LIN {X 0,Y 375.979,Z 740.463,A -85,B 0,C 180,E1 -12485.717,E2 -12485.717} C_VEL
LIN {X 0,Y 376.052,Z 740.601,A -85,B 0,C 180,E1 -12488.619,E2 -12488.619} C_VEL
LIN {X 0,Y 376.894,Z 745.86,A -85,B 0,C 180,E1 -12490.388,E2 -12490.388} C_VEL
LIN {X 0,Y 376.824,Z 753.026,A -85,B 0,C 180,E1 -12492.638,E2 -12492.638} C_VEL
LIN {X 0,Y 376.652,Z 755.465,A -85,B 0,C 180,E1 -12493.328,E2 -12493.328} C_VEL
LIN {X 0,Y 377.194,Z 758.566,A -85,B 0,C 180,E1 -12493.474,E2 -12493.474} C_VEL
LIN {X 0,Y 380.294,Z 775.584,A -85,B 0,C 180,E1 -12493.943,E2 -12493.943} C_VEL
LIN {X 0,Y 379.732,Z 831.118,A -85,B 0,C 180,E1 -12495.017,E2 -12495.017} C_VEL
LIN {X 0,Y 379.481,Z 840.948,A -85,B 0,C 180,E1 -12495.35,E2 -12495.35} C_VEL
LIN {X 0,Y 378.941,Z 852.061,A -85,B 0,C 180,E1 -12495.911,E2 -12495.911} C_VEL
LIN {X 0,Y 378.37,Z 862.886,A -85,B 0,C 180,E1 -12496.711,E2 -12496.711} C_VEL
LIN {X 0,Y 377.773,Z 871.277,A -85,B 0,C 180,E1 -12497.51,E2 -12497.51} C_VEL
LIN {X 0,Y 377.216,Z 879.195,A -85,B 0,C 180,E1 -12498.446,E2 -12498.446} C_VEL
LIN {X 0,Y 376.73,Z 884.882,A -85,B 0,C 180,E1 -12499.248,E2 -12499.248} C_VEL
LIN {X 0,Y 376.171,Z 891.229,A -85,B 0,C 180,E1 -12500.32,E2 -12500.32} C_VEL
LIN {X 0,Y 375.646,Z 897.671,A -85,B 0,C 180,E1 -12501.663,E2 -12501.663} C_VEL
LIN {X 0,Y 375.314,Z 902.635,A -85,B 0,C 180,E1 -12502.96,E2 -12502.96} C_VEL
LIN {X 0,Y 374.956,Z 907.561,A -85,B 0,C 180,E1 -12504.622,E2 -12504.622} C_VEL
LIN {X 0,Y 374.741,Z 909.88,A -85,B 0,C 180,E1 -12505.698,E2 -12505.698} C_VEL
LIN {X 0,Y 374.627,Z 911.643,A -85,B 0,C 180,E1 -12506.774,E2 -12506.774} C_VEL
LIN {X 0,Y 374.591,Z 912.912,A -85,B 0,C 180,E1 -12507.85,E2 -12507.85} C_VEL
LIN {X 0,Y 374.546,Z 913.715,A -85,B 0,C 180,E1 -12508.925,E2 -12508.925} C_VEL
LIN {X 0,Y 374.553,Z 914.02,A -85,B 0,C 180,E1 -12510,E2 -12510} C_VEL
LIN {X 0,Y 374.545,Z 913.744,A -85,B 0,C 180,E1 -12511.075,E2 -12511.075} C_VEL
LIN {X 0,Y 374.577,Z 913,A -85,B 0,C 180,E1 -12512.151,E2 -12512.151} C_VEL
LIN {X 0,Y 374.626,Z 911.789,A -85,B 0,C 180,E1 -12513.226,E2 -12513.226} C_VEL
LIN {X 0,Y 374.83,Z 908.942,A -85,B 0,C 180,E1 -12514.84,E2 -12514.84} C_VEL
LIN {X 0,Y 375.043,Z 906.351,A -85,B 0,C 180,E1 -12515.916,E2 -12515.916} C_VEL
LIN {X 0,Y 375.383,Z 901.251,A -85,B 0,C 180,E1 -12517.531,E2 -12517.531} C_VEL
LIN {X 0,Y 375.802,Z 895.762,A -85,B 0,C 180,E1 -12518.875,E2 -12518.875} C_VEL
LIN {X 0,Y 376.443,Z 888.863,A -85,B 0,C 180,E1 -12520.216,E2 -12520.216} C_VEL
LIN {X 0,Y 377.105,Z 880.938,A -85,B 0,C 180,E1 -12521.421,E2 -12521.421} C_VEL
LIN {X 0,Y 377.657,Z 873.381,A -85,B 0,C 180,E1 -12522.357,E2 -12522.357} C_VEL
LIN {X 0,Y 378.109,Z 866.955,A -85,B 0,C 180,E1 -12523.025,E2 -12523.025} C_VEL
LIN {X 0,Y 378.592,Z 859.142,A -85,B 0,C 180,E1 -12523.691,E2 -12523.691} C_VEL
LIN {X 0,Y 379.141,Z 850.18,A -85,B 0,C 180,E1 -12524.286,E2 -12524.286} C_VEL
LIN {X 0,Y 379.49,Z 840.834,A -85,B 0,C 180,E1 -12524.753,E2 -12524.753} C_VEL
LIN {X 0,Y 379.72,Z 831.346,A -85,B 0,C 180,E1 -12525.076,E2 -12525.076} C_VEL
LIN {X 0,Y 379.187,Z 825.564,A -85,B 0,C 180,E1 -12525.242,E2 -12525.242} C_VEL
LIN {X 0,Y 373.815,Z 806.862,A -85,B 0,C 180,E1 -12525.837,E2 -12525.837} C_VEL
LIN {X 0,Y 373.236,Z 801.048,A -85,B 0,C 180,E1 -12525.973,E2 -12525.973} C_VEL
LIN {X 0,Y 373.404,Z 775.423,A -85,B 0,C 180,E1 -12526.469,E2 -12526.469} C_VEL
LIN {X 0,Y 369.708,Z 755.57,A -85,B 0,C 180,E1 -12527.065,E2 -12527.065} C_VEL
LIN {X 0,Y 370.003,Z 748.159,A -85,B 0,C 180,E1 -12529.415,E2 -12529.415} C_VEL
LIN {X 0,Y 369.004,Z 741.425,A -85,B 0,C 180,E1 -12531.728,E2 -12531.728} C_VEL
LIN {X 0,Y 368.927,Z 741.344,A -85,B 0,C 180,E1 -12534.778,E2 -12534.778} C_VEL
LIN {X 0,Y 368.917,Z 741.343,A -85,B 0,C 180,E1 -12538.441,E2 -12538.441} C_VEL
LIN {X 0,Y 368.911,Z 741.334,A -85,B 0,C 180,E1 -12540.987,E2 -12540.987} C_VEL
LIN {X 0,Y 368.937,Z 741.344,A -85,B 0,C 180,E1 -12544.853,E2 -12544.853} C_VEL
LIN {X 0,Y 368.907,Z 741.323,A -85,B 0,C 180,E1 -12548.64,E2 -12548.64} C_VEL
LIN {X 0,Y 368.882,Z 741.346,A -85,B 0,C 180,E1 -12552.009,E2 -12552.009} C_VEL
LIN {X 0,Y 368.881,Z 741.332,A -85,B 0,C 180,E1 -12555.176,E2 -12555.176} C_VEL
LIN {X 0,Y 368.882,Z 741.305,A -85,B 0,C 180,E1 -12558.177,E2 -12558.177} C_VEL
LIN {X 0,Y 368.909,Z 741.34,A -85,B 0,C 180,E1 -12561.36,E2 -12561.36} C_VEL
LIN {X 0,Y 368.937,Z 741.334,A -85,B 0,C 180,E1 -12565.146,E2 -12565.146} C_VEL
LIN {X 0,Y 368.93,Z 741.342,A -85,B 0,C 180,E1 -12569.046,E2 -12569.046} C_VEL
LIN {X 0,Y 368.964,Z 741.329,A -85,B 0,C 180,E1 -12572.797,E2 -12572.797} C_VEL
LIN {X 0,Y 368.939,Z 741.332,A -85,B 0,C 180,E1 -12576.116,E2 -12576.116} C_VEL
LIN {X 0,Y 368.937,Z 741.335,A -85,B 0,C 180,E1 -12579.947,E2 -12579.947} C_VEL
LIN {X 0,Y 368.97,Z 741.32,A -85,B 0,C 180,E1 -12583.398,E2 -12583.398} C_VEL
LIN {X 0,Y 369.059,Z 741.323,A -85,B 0,C 180,E1 -12586.79,E2 -12586.79} C_VEL
LIN {X 0,Y 369.069,Z 741.314,A -85,B 0,C 180,E1 -12590.132,E2 -12590.132} C_VEL
LIN {X 0,Y 369.189,Z 741.283,A -85,B 0,C 180,E1 -12592.342,E2 -12592.342} C_VEL
LIN {X 0,Y 369.146,Z 741.303,A -85,B 0,C 180,E1 -12594.537,E2 -12594.537} C_VEL
LIN {X 0,Y 369.321,Z 741.292,A -85,B 0,C 180,E1 -12597.819,E2 -12597.819} C_VEL
LIN {X 0,Y 369.458,Z 741.265,A -85,B 0,C 180,E1 -12600,E2 -12600} C_VEL
LIN {X 0,Y 369.318,Z 741.268,A -85,B 0,C 180,E1 -12602.181,E2 -12602.181} C_VEL
LIN {X 0,Y 369.201,Z 741.305,A -85,B 0,C 180,E1 -12606.558,E2 -12606.558} C_VEL
LIN {X 0,Y 369.069,Z 741.316,A -85,B 0,C 180,E1 -12609.868,E2 -12609.868} C_VEL
LIN {X 0,Y 369.038,Z 741.314,A -85,B 0,C 180,E1 -12613.772,E2 -12613.772} C_VEL
LIN {X 0,Y 369.002,Z 741.335,A -85,B 0,C 180,E1 -12617.768,E2 -12617.768} C_VEL
LIN {X 0,Y 368.942,Z 741.321,A -85,B 0,C 180,E1 -12621.219,E2 -12621.219} C_VEL
LIN {X 0,Y 368.959,Z 741.336,A -85,B 0,C 180,E1 -12624.775,E2 -12624.775} C_VEL
LIN {X 0,Y 368.964,Z 741.332,A -85,B 0,C 180,E1 -12627.203,E2 -12627.203} C_VEL
LIN {X 0,Y 368.93,Z 741.335,A -85,B 0,C 180,E1 -12630.953,E2 -12630.953} C_VEL
LIN {X 0,Y 368.93,Z 741.334,A -85,B 0,C 180,E1 -12635.001,E2 -12635.001} C_VEL
LIN {X 0,Y 368.913,Z 741.297,A -85,B 0,C 180,E1 -12638.641,E2 -12638.641} C_VEL
LIN {X 0,Y 368.91,Z 741.325,A -85,B 0,C 180,E1 -12641.818,E2 -12641.818} C_VEL
LIN {X 0,Y 368.881,Z 741.345,A -85,B 0,C 180,E1 -12645.176,E2 -12645.176} C_VEL
LIN {X 0,Y 368.883,Z 741.331,A -85,B 0,C 180,E1 -12648.178,E2 -12648.178} C_VEL
LIN {X 0,Y 368.912,Z 741.343,A -85,B 0,C 180,E1 -12651.359,E2 -12651.359} C_VEL
LIN {X 0,Y 368.937,Z 741.339,A -85,B 0,C 180,E1 -12655.146,E2 -12655.146} C_VEL
LIN {X 0,Y 368.929,Z 741.318,A -85,B 0,C 180,E1 -12659.046,E2 -12659.046} C_VEL
LIN {X 0,Y 368.98,Z 741.337,A -85,B 0,C 180,E1 -12661.564,E2 -12661.564} C_VEL
LIN {X 0,Y 369.024,Z 741.491,A -85,B 0,C 180,E1 -12663.59,E2 -12663.59} C_VEL
LIN {X 0,Y 370.89,Z 751.613,A -85,B 0,C 180,E1 -12666.551,E2 -12666.551} C_VEL
LIN {X 0,Y 371.176,Z 754.872,A -85,B 0,C 180,E1 -12667.454,E2 -12667.454} C_VEL
LIN {X 0,Y 369.878,Z 770.415,A -85,B 0,C 180,E1 -12671.597,E2 -12671.597} C_VEL
LIN {X 0,Y 369.516,Z 775.616,A -85,B 0,C 180,E1 -12672.926,E2 -12672.926} C_VEL
LIN {X 0,Y 370.037,Z 779.164,A -85,B 0,C 180,E1 -12673.08,E2 -12673.08} C_VEL
LIN {X 0,Y 373.258,Z 802.94,A -85,B 0,C 180,E1 -12673.696,E2 -12673.696} C_VEL
LIN {X 0,Y 372.715,Z 853.211,A -85,B 0,C 180,E1 -12674.693,E2 -12674.693} C_VEL
LIN {X 0,Y 372.288,Z 863.626,A -85,B 0,C 180,E1 -12675.06,E2 -12675.06} C_VEL
LIN {X 0,Y 371.713,Z 874.301,A -85,B 0,C 180,E1 -12675.632,E2 -12675.632} C_VEL
LIN {X 0,Y 371.026,Z 884.916,A -85,B 0,C 180,E1 -12676.443,E2 -12676.443} C_VEL
LIN {X 0,Y 370.362,Z 893.234,A -85,B 0,C 180,E1 -12677.256,E2 -12677.256} C_VEL
LIN {X 0,Y 369.716,Z 901.108,A -85,B 0,C 180,E1 -12678.209,E2 -12678.209} C_VEL
LIN {X 0,Y 369.106,Z 908.473,A -85,B 0,C 180,E1 -12679.301,E2 -12679.301} C_VEL
LIN {X 0,Y 368.504,Z 915.947,A -85,B 0,C 180,E1 -12680.671,E2 -12680.671} C_VEL
LIN {X 0,Y 367.943,Z 922.772,A -85,B 0,C 180,E1 -12682.316,E2 -12682.316} C_VEL
LIN {X 0,Y 367.662,Z 927.276,A -85,B 0,C 180,E1 -12683.719,E2 -12683.719} C_VEL
LIN {X 0,Y 367.569,Z 930.612,A -85,B 0,C 180,E1 -12685.064,E2 -12685.064} C_VEL
LIN {X 0,Y 367.4,Z 933.52,A -85,B 0,C 180,E1 -12686.71,E2 -12686.71} C_VEL
LIN {X 0,Y 367.361,Z 934.775,A -85,B 0,C 180,E1 -12687.807,E2 -12687.807} C_VEL
LIN {X 0,Y 367.415,Z 935.557,A -85,B 0,C 180,E1 -12688.904,E2 -12688.904} C_VEL
LIN {X 0,Y 367.454,Z 935.854,A -85,B 0,C 180,E1 -12690,E2 -12690} C_VEL
LIN {X 0,Y 367.415,Z 935.555,A -85,B 0,C 180,E1 -12691.096,E2 -12691.096} C_VEL
LIN {X 0,Y 367.362,Z 934.767,A -85,B 0,C 180,E1 -12692.193,E2 -12692.193} C_VEL
LIN {X 0,Y 367.4,Z 933.507,A -85,B 0,C 180,E1 -12693.29,E2 -12693.29} C_VEL
LIN {X 0,Y 367.569,Z 930.594,A -85,B 0,C 180,E1 -12694.936,E2 -12694.936} C_VEL
LIN {X 0,Y 367.662,Z 927.254,A -85,B 0,C 180,E1 -12696.281,E2 -12696.281} C_VEL
LIN {X 0,Y 368.035,Z 921.778,A -85,B 0,C 180,E1 -12697.958,E2 -12697.958} C_VEL
LIN {X 0,Y 368.491,Z 915.9,A -85,B 0,C 180,E1 -12699.33,E2 -12699.33} C_VEL
LIN {X 0,Y 369.105,Z 908.424,A -85,B 0,C 180,E1 -12700.699,E2 -12700.699} C_VEL
LIN {X 0,Y 369.715,Z 901.052,A -85,B 0,C 180,E1 -12701.791,E2 -12701.791} C_VEL
LIN {X 0,Y 370.362,Z 893.16,A -85,B 0,C 180,E1 -12702.744,E2 -12702.744} C_VEL
LIN {X 0,Y 371.042,Z 884.824,A -85,B 0,C 180,E1 -12703.556,E2 -12703.556} C_VEL
LIN {X 0,Y 371.72,Z 874.174,A -85,B 0,C 180,E1 -12704.368,E2 -12704.368} C_VEL
LIN {X 0,Y 372.284,Z 862.584,A -85,B 0,C 180,E1 -12704.975,E2 -12704.975} C_VEL
LIN {X 0,Y 372.712,Z 852.881,A -85,B 0,C 180,E1 -12705.307,E2 -12705.307} C_VEL
LIN {X 0,Y 373.256,Z 802.524,A -85,B 0,C 180,E1 -12706.303,E2 -12706.303} C_VEL
LIN {X 0,Y 369.55,Z 776.321,A -85,B 0,C 180,E1 -12707.005,E2 -12707.005} C_VEL
LIN {X 0,Y 369.518,Z 775.227,A -85,B 0,C 180,E1 -12707.146,E2 -12707.146} C_VEL
LIN {X 0,Y 370.392,Z 763.413,A -85,B 0,C 180,E1 -12710.26,E2 -12710.26} C_VEL
LIN {X 0,Y 371.159,Z 753.751,A -85,B 0,C 180,E1 -12712.841,E2 -12712.841} C_VEL
LIN {X 0,Y 369.715,Z 745.091,A -85,B 0,C 180,E1 -12715.322,E2 -12715.322} C_VEL
LIN {X 0,Y 368.989,Z 741.357,A -85,B 0,C 180,E1 -12716.493,E2 -12716.493} C_VEL
LIN {X 0,Y 368.919,Z 741.326,A -85,B 0,C 180,E1 -12719.69,E2 -12719.69} C_VEL
LIN {X 0,Y 368.899,Z 741.344,A -85,B 0,C 180,E1 -12723.044,E2 -12723.044} C_VEL
LIN {X 0,Y 368.919,Z 741.335,A -85,B 0,C 180,E1 -12726.197,E2 -12726.197} C_VEL
LIN {X 0,Y 368.906,Z 741.345,A -85,B 0,C 180,E1 -12728.953,E2 -12728.953} C_VEL
LIN {X 0,Y 368.882,Z 741.333,A -85,B 0,C 180,E1 -12732.01,E2 -12732.01} C_VEL
LIN {X 0,Y 368.881,Z 741.348,A -85,B 0,C 180,E1 -12735.176,E2 -12735.176} C_VEL
LIN {X 0,Y 368.91,Z 741.323,A -85,B 0,C 180,E1 -12738.182,E2 -12738.182} C_VEL
LIN {X 0,Y 368.913,Z 741.297,A -85,B 0,C 180,E1 -12741.359,E2 -12741.359} C_VEL
LIN {X 0,Y 368.938,Z 741.334,A -85,B 0,C 180,E1 -12745.147,E2 -12745.147} C_VEL
LIN {X 0,Y 368.93,Z 741.334,A -85,B 0,C 180,E1 -12749.047,E2 -12749.047} C_VEL
LIN {X 0,Y 368.964,Z 741.333,A -85,B 0,C 180,E1 -12752.797,E2 -12752.797} C_VEL
LIN {X 0,Y 368.946,Z 741.335,A -85,B 0,C 180,E1 -12756.113,E2 -12756.113} C_VEL
LIN {X 0,Y 368.946,Z 741.326,A -85,B 0,C 180,E1 -12759.948,E2 -12759.948} C_VEL
LIN {X 0,Y 368.978,Z 741.333,A -85,B 0,C 180,E1 -12763.399,E2 -12763.399} C_VEL
LIN {X 0,Y 369.059,Z 741.305,A -85,B 0,C 180,E1 -12766.79,E2 -12766.79} C_VEL
LIN {X 0,Y 369.069,Z 741.316,A -85,B 0,C 180,E1 -12770.132,E2 -12770.132} C_VEL
LIN {X 0,Y 369.201,Z 741.304,A -85,B 0,C 180,E1 -12773.442,E2 -12773.442} C_VEL
LIN {X 0,Y 369.319,Z 741.268,A -85,B 0,C 180,E1 -12777.819,E2 -12777.819} C_VEL
LIN {X 0,Y 369.46,Z 741.264,A -85,B 0,C 180,E1 -12780,E2 -12780} C_VEL
LIN {X 0,Y 369.321,Z 741.291,A -85,B 0,C 180,E1 -12782.181,E2 -12782.181} C_VEL
LIN {X 0,Y 369.209,Z 741.288,A -85,B 0,C 180,E1 -12786.558,E2 -12786.558} C_VEL
LIN {X 0,Y 369.139,Z 741.298,A -85,B 0,C 180,E1 -12788.761,E2 -12788.761} C_VEL
LIN {X 0,Y 369.007,Z 741.329,A -85,B 0,C 180,E1 -12792.093,E2 -12792.093} C_VEL
LIN {X 0,Y 368.999,Z 741.32,A -85,B 0,C 180,E1 -12795.465,E2 -12795.465} C_VEL
LIN {X 0,Y 368.956,Z 741.327,A -85,B 0,C 180,E1 -12798.894,E2 -12798.894} C_VEL
LIN {X 0,Y 368.924,Z 741.341,A -85,B 0,C 180,E1 -12802.396,E2 -12802.396} C_VEL
LIN {X 0,Y 369.001,Z 741.313,A -85,B 0,C 180,E1 -12805.98,E2 -12805.98} C_VEL
LIN {X 0,Y 368.916,Z 741.342,A -85,B 0,C 180,E1 -12809.69,E2 -12809.69} C_VEL
LIN {X 0,Y 368.898,Z 741.335,A -85,B 0,C 180,E1 -12813.043,E2 -12813.043} C_VEL
LIN {X 0,Y 368.918,Z 741.34,A -85,B 0,C 180,E1 -12816.197,E2 -12816.197} C_VEL
LIN {X 0,Y 368.904,Z 741.34,A -85,B 0,C 180,E1 -12818.953,E2 -12818.953} C_VEL
LIN {X 0,Y 368.88,Z 741.304,A -85,B 0,C 180,E1 -12822.009,E2 -12822.009} C_VEL
LIN {X 0,Y 368.881,Z 741.333,A -85,B 0,C 180,E1 -12825.176,E2 -12825.176} C_VEL
LIN {X 0,Y 368.884,Z 741.345,A -85,B 0,C 180,E1 -12828.178,E2 -12828.178} C_VEL
LIN {X 0,Y 368.908,Z 741.323,A -85,B 0,C 180,E1 -12831.36,E2 -12831.36} C_VEL
LIN {X 0,Y 368.937,Z 741.343,A -85,B 0,C 180,E1 -12835.147,E2 -12835.147} C_VEL
LIN {X 0,Y 368.93,Z 741.33,A -85,B 0,C 180,E1 -12839.047,E2 -12839.047} C_VEL
LIN {X 0,Y 368.876,Z 741.348,A -85,B 0,C 180,E1 -12842.79,E2 -12842.79} C_VEL
LIN {X 0,Y 368.929,Z 741.337,A -85,B 0,C 180,E1 -12846.119,E2 -12846.119} C_VEL
LIN {X 0,Y 369.008,Z 741.476,A -85,B 0,C 180,E1 -12848.419,E2 -12848.419} C_VEL
LIN {X 0,Y 369.972,Z 747.844,A -85,B 0,C 180,E1 -12850.584,E2 -12850.584} C_VEL
LIN {X 0,Y 369.74,Z 755.365,A -85,B 0,C 180,E1 -12852.943,E2 -12852.943} C_VEL
LIN {X 0,Y 369.758,Z 756.158,A -85,B 0,C 180,E1 -12853.061,E2 -12853.061} C_VEL
LIN {X 0,Y 373.52,Z 776.553,A -85,B 0,C 180,E1 -12853.658,E2 -12853.658} C_VEL
LIN {X 0,Y 372.894,Z 831.345,A -85,B 0,C 180,E1 -12854.736,E2 -12854.736} C_VEL
LIN {X 0,Y 372.685,Z 840.337,A -85,B 0,C 180,E1 -12855.042,E2 -12855.042} C_VEL
LIN {X 0,Y 372.198,Z 849.88,A -85,B 0,C 180,E1 -12855.511,E2 -12855.511} C_VEL
LIN {X 0,Y 371.693,Z 859.886,A -85,B 0,C 180,E1 -12856.189,E2 -12856.189} C_VEL
LIN {X 0,Y 370.932,Z 870.264,A -85,B 0,C 180,E1 -12857.137,E2 -12857.137} C_VEL
LIN {X 0,Y 370.33,Z 878.39,A -85,B 0,C 180,E1 -12858.09,E2 -12858.09} C_VEL
LIN {X 0,Y 369.767,Z 885.094,A -85,B 0,C 180,E1 -12859.043,E2 -12859.043} C_VEL
LIN {X 0,Y 369.19,Z 891.44,A -85,B 0,C 180,E1 -12860.135,E2 -12860.135} C_VEL
LIN {X 0,Y 368.614,Z 897.882,A -85,B 0,C 180,E1 -12861.503,E2 -12861.503} C_VEL
LIN {X 0,Y 368.259,Z 903.202,A -85,B 0,C 180,E1 -12862.928,E2 -12862.928} C_VEL
LIN {X 0,Y 367.91,Z 907.77,A -85,B 0,C 180,E1 -12864.519,E2 -12864.519} C_VEL
LIN {X 0,Y 367.675,Z 910.089,A -85,B 0,C 180,E1 -12865.615,E2 -12865.615} C_VEL
LIN {X 0,Y 367.54,Z 911.852,A -85,B 0,C 180,E1 -12866.711,E2 -12866.711} C_VEL
LIN {X 0,Y 367.495,Z 913.122,A -85,B 0,C 180,E1 -12867.808,E2 -12867.808} C_VEL
LIN {X 0,Y 367.45,Z 913.924,A -85,B 0,C 180,E1 -12868.904,E2 -12868.904} C_VEL
LIN {X 0,Y 367.456,Z 914.229,A -85,B 0,C 180,E1 -12870,E2 -12870} C_VEL
LIN {X 0,Y 367.449,Z 913.952,A -85,B 0,C 180,E1 -12871.096,E2 -12871.096} C_VEL
LIN {X 0,Y 367.482,Z 913.208,A -85,B 0,C 180,E1 -12872.192,E2 -12872.192} C_VEL
LIN {X 0,Y 367.539,Z 911.997,A -85,B 0,C 180,E1 -12873.289,E2 -12873.289} C_VEL
LIN {X 0,Y 367.776,Z 909.15,A -85,B 0,C 180,E1 -12874.933,E2 -12874.933} C_VEL
LIN {X 0,Y 367.99,Z 906.558,A -85,B 0,C 180,E1 -12876.03,E2 -12876.03} C_VEL
LIN {X 0,Y 368.276,Z 902.6,A -85,B 0,C 180,E1 -12877.346,E2 -12877.346} C_VEL
LIN {X 0,Y 368.563,Z 898.305,A -85,B 0,C 180,E1 -12878.498,E2 -12878.498} C_VEL
LIN {X 0,Y 369.013,Z 893.361,A -85,B 0,C 180,E1 -12879.593,E2 -12879.593} C_VEL
LIN {X 0,Y 369.604,Z 887.392,A -85,B 0,C 180,E1 -12880.684,E2 -12880.684} C_VEL
LIN {X 0,Y 370.239,Z 880.125,A -85,B 0,C 180,E1 -12881.774,E2 -12881.774} C_VEL
LIN {X 0,Y 370.743,Z 873.585,A -85,B 0,C 180,E1 -12882.592,E2 -12882.592} C_VEL
LIN {X 0,Y 371.222,Z 867.158,A -85,B 0,C 180,E1 -12883.271,E2 -12883.271} C_VEL
LIN {X 0,Y 371.722,Z 859.343,A -85,B 0,C 180,E1 -12883.949,E2 -12883.949} C_VEL
LIN {X 0,Y 372.276,Z 850.38,A -85,B 0,C 180,E1 -12884.556,E2 -12884.556} C_VEL
LIN {X 0,Y 372.64,Z 841.03,A -85,B 0,C 180,E1 -12885.03,E2 -12885.03} C_VEL
LIN {X 0,Y 372.89,Z 831.244,A -85,B 0,C 180,E1 -12885.366,E2 -12885.366} C_VEL
LIN {X 0,Y 373.236,Z 801.048,A -85,B 0,C 180,E1 -12885.973,E2 -12885.973} C_VEL
LIN {X 0,Y 372.713,Z 795.23,A -85,B 0,C 180,E1 -12886.111,E2 -12886.111} C_VEL
LIN {X 0,Y 370.117,Z 785.876,A -85,B 0,C 180,E1 -12886.414,E2 -12886.414} C_VEL
LIN {X 0,Y 367.565,Z 778.467,A -85,B 0,C 180,E1 -12886.681,E2 -12886.681} C_VEL
LIN {X 0,Y 365.646,Z 770.867,A -85,B 0,C 180,E1 -12886.925,E2 -12886.925} C_VEL
LIN {X 0,Y 362.776,Z 755.777,A -85,B 0,C 180,E1 -12887.402,E2 -12887.402} C_VEL
LIN {X 0,Y 363.005,Z 750.14,A -85,B 0,C 180,E1 -12889.216,E2 -12889.216} C_VEL
LIN {X 0,Y 362.24,Z 743.79,A -85,B 0,C 180,E1 -12891.366,E2 -12891.366} C_VEL
LIN {X 0,Y 361.954,Z 742.299,A -85,B 0,C 180,E1 -12891.949,E2 -12891.949} C_VEL
LIN {X 0,Y 361.884,Z 742.22,A -85,B 0,C 180,E1 -12895.293,E2 -12895.293} C_VEL
LIN {X 0,Y 361.856,Z 742.222,A -85,B 0,C 180,E1 -12899.074,E2 -12899.074} C_VEL
LIN {X 0,Y 361.849,Z 742.217,A -85,B 0,C 180,E1 -12902.945,E2 -12902.945} C_VEL
LIN {X 0,Y 361.869,Z 742.222,A -85,B 0,C 180,E1 -12905.637,E2 -12905.637} C_VEL
LIN {X 0,Y 361.868,Z 742.201,A -85,B 0,C 180,E1 -12909.026,E2 -12909.026} C_VEL
LIN {X 0,Y 361.837,Z 742.226,A -85,B 0,C 180,E1 -12912.829,E2 -12912.829} C_VEL
LIN {X 0,Y 361.819,Z 742.202,A -85,B 0,C 180,E1 -12915.947,E2 -12915.947} C_VEL
LIN {X 0,Y 361.835,Z 742.198,A -85,B 0,C 180,E1 -12919.245,E2 -12919.245} C_VEL
LIN {X 0,Y 361.864,Z 742.223,A -85,B 0,C 180,E1 -12922.777,E2 -12922.777} C_VEL
LIN {X 0,Y 361.855,Z 742.212,A -85,B 0,C 180,E1 -12925.72,E2 -12925.72} C_VEL
LIN {X 0,Y 361.874,Z 742.218,A -85,B 0,C 180,E1 -12929.672,E2 -12929.672} C_VEL
LIN {X 0,Y 361.955,Z 742.193,A -85,B 0,C 180,E1 -12933.475,E2 -12933.475} C_VEL
LIN {X 0,Y 361.884,Z 742.219,A -85,B 0,C 180,E1 -12937.144,E2 -12937.144} C_VEL
LIN {X 0,Y 361.905,Z 742.213,A -85,B 0,C 180,E1 -12940.723,E2 -12940.723} C_VEL
LIN {X 0,Y 361.945,Z 742.198,A -85,B 0,C 180,E1 -12944.226,E2 -12944.226} C_VEL
LIN {X 0,Y 362,Z 742.201,A -85,B 0,C 180,E1 -12946.528,E2 -12946.528} C_VEL
LIN {X 0,Y 362.033,Z 742.191,A -85,B 0,C 180,E1 -12949.938,E2 -12949.938} C_VEL
LIN {X 0,Y 362.152,Z 742.159,A -85,B 0,C 180,E1 -12952.192,E2 -12952.192} C_VEL
LIN {X 0,Y 362.119,Z 742.178,A -85,B 0,C 180,E1 -12954.431,E2 -12954.431} C_VEL
LIN {X 0,Y 362.285,Z 742.168,A -85,B 0,C 180,E1 -12957.776,E2 -12957.776} C_VEL
LIN {X 0,Y 362.428,Z 742.14,A -85,B 0,C 180,E1 -12960,E2 -12960} C_VEL
LIN {X 0,Y 362.282,Z 742.144,A -85,B 0,C 180,E1 -12962.223,E2 -12962.223} C_VEL
LIN {X 0,Y 362.163,Z 742.181,A -85,B 0,C 180,E1 -12966.686,E2 -12966.686} C_VEL
LIN {X 0,Y 362.033,Z 742.19,A -85,B 0,C 180,E1 -12970.062,E2 -12970.062} C_VEL
LIN {X 0,Y 361.999,Z 742.192,A -85,B 0,C 180,E1 -12973.899,E2 -12973.899} C_VEL
LIN {X 0,Y 361.969,Z 742.208,A -85,B 0,C 180,E1 -12977.939,E2 -12977.939} C_VEL
LIN {X 0,Y 361.899,Z 742.199,A -85,B 0,C 180,E1 -12981.652,E2 -12981.652} C_VEL
LIN {X 0,Y 361.929,Z 742.211,A -85,B 0,C 180,E1 -12985.29,E2 -12985.29} C_VEL
LIN {X 0,Y 361.909,Z 742.211,A -85,B 0,C 180,E1 -12987.779,E2 -12987.779} C_VEL
LIN {X 0,Y 361.838,Z 742.22,A -85,B 0,C 180,E1 -12991.629,E2 -12991.629} C_VEL
LIN {X 0,Y 361.875,Z 742.213,A -85,B 0,C 180,E1 -12995.345,E2 -12995.345} C_VEL
LIN {X 0,Y 361.874,Z 742.17,A -85,B 0,C 180,E1 -12999.027,E2 -12999.027} C_VEL
LIN {X 0,Y 361.857,Z 742.209,A -85,B 0,C 180,E1 -13002.435,E2 -13002.435} C_VEL
LIN {X 0,Y 361.82,Z 742.227,A -85,B 0,C 180,E1 -13005.946,E2 -13005.946} C_VEL
LIN {X 0,Y 361.837,Z 742.21,A -85,B 0,C 180,E1 -13009.244,E2 -13009.244} C_VEL
LIN {X 0,Y 361.872,Z 742.217,A -85,B 0,C 180,E1 -13012.775,E2 -13012.775} C_VEL
LIN {X 0,Y 361.855,Z 742.222,A -85,B 0,C 180,E1 -13015.72,E2 -13015.72} C_VEL
LIN {X 0,Y 361.875,Z 742.196,A -85,B 0,C 180,E1 -13019.672,E2 -13019.672} C_VEL
LIN {X 0,Y 361.961,Z 742.256,A -85,B 0,C 180,E1 -13023.272,E2 -13023.272} C_VEL
LIN {X 0,Y 363.652,Z 751.413,A -85,B 0,C 180,E1 -13026.056,E2 -13026.056} C_VEL
LIN {X 0,Y 364.221,Z 755.766,A -85,B 0,C 180,E1 -13027.299,E2 -13027.299} C_VEL
LIN {X 0,Y 362.922,Z 770.518,A -85,B 0,C 180,E1 -13031.314,E2 -13031.314} C_VEL
LIN {X 0,Y 362.529,Z 775.411,A -85,B 0,C 180,E1 -13032.586,E2 -13032.586} C_VEL
LIN {X 0,Y 363.091,Z 779.315,A -85,B 0,C 180,E1 -13032.754,E2 -13032.754} C_VEL
LIN {X 0,Y 366.414,Z 802.912,A -85,B 0,C 180,E1 -13033.386,E2 -13033.386} C_VEL
LIN {X 0,Y 365.905,Z 852.126,A -85,B 0,C 180,E1 -13034.377,E2 -13034.377} C_VEL
LIN {X 0,Y 365.509,Z 861.763,A -85,B 0,C 180,E1 -13034.705,E2 -13034.705} C_VEL
LIN {X 0,Y 364.987,Z 871.803,A -85,B 0,C 180,E1 -13035.218,E2 -13035.218} C_VEL
LIN {X 0,Y 364.233,Z 883.208,A -85,B 0,C 180,E1 -13036.043,E2 -13036.043} C_VEL
LIN {X 0,Y 363.547,Z 891.797,A -85,B 0,C 180,E1 -13036.871,E2 -13036.871} C_VEL
LIN {X 0,Y 362.827,Z 899.878,A -85,B 0,C 180,E1 -13037.84,E2 -13037.84} C_VEL
LIN {X 0,Y 362.271,Z 906.557,A -85,B 0,C 180,E1 -13038.814,E2 -13038.814} C_VEL
LIN {X 0,Y 361.697,Z 912.898,A -85,B 0,C 180,E1 -13039.929,E2 -13039.929} C_VEL
LIN {X 0,Y 361.253,Z 918.168,A -85,B 0,C 180,E1 -13041.046,E2 -13041.046} C_VEL
LIN {X 0,Y 360.909,Z 922.565,A -85,B 0,C 180,E1 -13042.166,E2 -13042.166} C_VEL
LIN {X 0,Y 360.556,Z 927.548,A -85,B 0,C 180,E1 -13043.771,E2 -13043.771} C_VEL
LIN {X 0,Y 360.465,Z 930.403,A -85,B 0,C 180,E1 -13044.967,E2 -13044.967} C_VEL
LIN {X 0,Y 360.323,Z 933.312,A -85,B 0,C 180,E1 -13046.645,E2 -13046.645} C_VEL
LIN {X 0,Y 360.267,Z 934.566,A -85,B 0,C 180,E1 -13047.764,E2 -13047.764} C_VEL
LIN {X 0,Y 360.314,Z 935.349,A -85,B 0,C 180,E1 -13048.882,E2 -13048.882} C_VEL
LIN {X 0,Y 360.357,Z 935.645,A -85,B 0,C 180,E1 -13050,E2 -13050} C_VEL
LIN {X 0,Y 360.314,Z 935.346,A -85,B 0,C 180,E1 -13051.118,E2 -13051.118} C_VEL
LIN {X 0,Y 360.267,Z 934.558,A -85,B 0,C 180,E1 -13052.236,E2 -13052.236} C_VEL
LIN {X 0,Y 360.323,Z 933.298,A -85,B 0,C 180,E1 -13053.355,E2 -13053.355} C_VEL
LIN {X 0,Y 360.465,Z 930.384,A -85,B 0,C 180,E1 -13055.033,E2 -13055.033} C_VEL
LIN {X 0,Y 360.556,Z 927.524,A -85,B 0,C 180,E1 -13056.229,E2 -13056.229} C_VEL
LIN {X 0,Y 360.909,Z 922.531,A -85,B 0,C 180,E1 -13057.834,E2 -13057.834} C_VEL
LIN {X 0,Y 361.463,Z 915.688,A -85,B 0,C 180,E1 -13059.513,E2 -13059.513} C_VEL
LIN {X 0,Y 362.104,Z 908.211,A -85,B 0,C 180,E1 -13060.908,E2 -13060.908} C_VEL
LIN {X 0,Y 362.748,Z 900.84,A -85,B 0,C 180,E1 -13062.021,E2 -13062.021} C_VEL
LIN {X 0,Y 363.413,Z 892.947,A -85,B 0,C 180,E1 -13062.992,E2 -13062.992} C_VEL
LIN {X 0,Y 364.143,Z 884.611,A -85,B 0,C 180,E1 -13063.818,E2 -13063.818} C_VEL
LIN {X 0,Y 364.856,Z 873.96,A -85,B 0,C 180,E1 -13064.644,E2 -13064.644} C_VEL
LIN {X 0,Y 365.435,Z 862.366,A -85,B 0,C 180,E1 -13065.262,E2 -13065.262} C_VEL
LIN {X 0,Y 365.876,Z 852.658,A -85,B 0,C 180,E1 -13065.6,E2 -13065.6} C_VEL
LIN {X 0,Y 366.317,Z 802.202,A -85,B 0,C 180,E1 -13066.623,E2 -13066.623} C_VEL
LIN {X 0,Y 362.588,Z 776.132,A -85,B 0,C 180,E1 -13067.341,E2 -13067.341} C_VEL
LIN {X 0,Y 362.552,Z 775.019,A -85,B 0,C 180,E1 -13067.486,E2 -13067.486} C_VEL
LIN {X 0,Y 363.708,Z 761.086,A -85,B 0,C 180,E1 -13071.242,E2 -13071.242} C_VEL
LIN {X 0,Y 364.162,Z 754.645,A -85,B 0,C 180,E1 -13073.005,E2 -13073.005} C_VEL
LIN {X 0,Y 362.452,Z 744.898,A -85,B 0,C 180,E1 -13075.867,E2 -13075.867} C_VEL
LIN {X 0,Y 361.96,Z 742.231,A -85,B 0,C 180,E1 -13076.744,E2 -13076.744} C_VEL
LIN {X 0,Y 361.875,Z 742.197,A -85,B 0,C 180,E1 -13080.328,E2 -13080.328} C_VEL
LIN {X 0,Y 361.855,Z 742.223,A -85,B 0,C 180,E1 -13084.28,E2 -13084.28} C_VEL
LIN {X 0,Y 361.872,Z 742.217,A -85,B 0,C 180,E1 -13087.225,E2 -13087.225} C_VEL
LIN {X 0,Y 361.837,Z 742.209,A -85,B 0,C 180,E1 -13090.756,E2 -13090.756} C_VEL
LIN {X 0,Y 361.818,Z 742.225,A -85,B 0,C 180,E1 -13094.368,E2 -13094.368} C_VEL
LIN {X 0,Y 361.857,Z 742.208,A -85,B 0,C 180,E1 -13097.565,E2 -13097.565} C_VEL
LIN {X 0,Y 361.874,Z 742.169,A -85,B 0,C 180,E1 -13100.973,E2 -13100.973} C_VEL
LIN {X 0,Y 361.875,Z 742.213,A -85,B 0,C 180,E1 -13104.655,E2 -13104.655} C_VEL
LIN {X 0,Y 361.838,Z 742.219,A -85,B 0,C 180,E1 -13108.371,E2 -13108.371} C_VEL
LIN {X 0,Y 361.909,Z 742.212,A -85,B 0,C 180,E1 -13112.221,E2 -13112.221} C_VEL
LIN {X 0,Y 361.929,Z 742.211,A -85,B 0,C 180,E1 -13114.71,E2 -13114.71} C_VEL
LIN {X 0,Y 361.899,Z 742.199,A -85,B 0,C 180,E1 -13118.348,E2 -13118.348} C_VEL
LIN {X 0,Y 361.969,Z 742.208,A -85,B 0,C 180,E1 -13122.061,E2 -13122.061} C_VEL
LIN {X 0,Y 361.999,Z 742.192,A -85,B 0,C 180,E1 -13126.101,E2 -13126.101} C_VEL
LIN {X 0,Y 362.033,Z 742.19,A -85,B 0,C 180,E1 -13129.938,E2 -13129.938} C_VEL
LIN {X 0,Y 362.163,Z 742.181,A -85,B 0,C 180,E1 -13133.314,E2 -13133.314} C_VEL
LIN {X 0,Y 362.283,Z 742.143,A -85,B 0,C 180,E1 -13137.777,E2 -13137.777} C_VEL
LIN {X 0,Y 362.43,Z 742.14,A -85,B 0,C 180,E1 -13140,E2 -13140} C_VEL
LIN {X 0,Y 362.285,Z 742.168,A -85,B 0,C 180,E1 -13142.224,E2 -13142.224} C_VEL
LIN {X 0,Y 362.173,Z 742.162,A -85,B 0,C 180,E1 -13146.686,E2 -13146.686} C_VEL
LIN {X 0,Y 362.076,Z 742.18,A -85,B 0,C 180,E1 -13148.933,E2 -13148.933} C_VEL
LIN {X 0,Y 361.962,Z 742.209,A -85,B 0,C 180,E1 -13152.332,E2 -13152.332} C_VEL
LIN {X 0,Y 361.963,Z 742.206,A -85,B 0,C 180,E1 -13154.62,E2 -13154.62} C_VEL
LIN {X 0,Y 361.912,Z 742.197,A -85,B 0,C 180,E1 -13158.102,E2 -13158.102} C_VEL
LIN {X 0,Y 361.862,Z 742.22,A -85,B 0,C 180,E1 -13161.655,E2 -13161.655} C_VEL
LIN {X 0,Y 361.928,Z 742.197,A -85,B 0,C 180,E1 -13165.29,E2 -13165.29} C_VEL
LIN {X 0,Y 361.91,Z 742.211,A -85,B 0,C 180,E1 -13167.779,E2 -13167.779} C_VEL
LIN {X 0,Y 361.838,Z 742.218,A -85,B 0,C 180,E1 -13171.629,E2 -13171.629} C_VEL
LIN {X 0,Y 361.875,Z 742.218,A -85,B 0,C 180,E1 -13175.345,E2 -13175.345} C_VEL
LIN {X 0,Y 361.87,Z 742.215,A -85,B 0,C 180,E1 -13179.027,E2 -13179.027} C_VEL
LIN {X 0,Y 361.836,Z 742.179,A -85,B 0,C 180,E1 -13182.829,E2 -13182.829} C_VEL
LIN {X 0,Y 361.82,Z 742.224,A -85,B 0,C 180,E1 -13185.947,E2 -13185.947} C_VEL
LIN {X 0,Y 361.837,Z 742.222,A -85,B 0,C 180,E1 -13189.245,E2 -13189.245} C_VEL
LIN {X 0,Y 361.864,Z 742.208,A -85,B 0,C 180,E1 -13192.777,E2 -13192.777} C_VEL
LIN {X 0,Y 361.855,Z 742.226,A -85,B 0,C 180,E1 -13195.72,E2 -13195.72} C_VEL
LIN {X 0,Y 361.866,Z 742.216,A -85,B 0,C 180,E1 -13199.671,E2 -13199.671} C_VEL
LIN {X 0,Y 361.875,Z 742.223,A -85,B 0,C 180,E1 -13203.469,E2 -13203.469} C_VEL
LIN {X 0,Y 361.889,Z 742.214,A -85,B 0,C 180,E1 -13207.145,E2 -13207.145} C_VEL
LIN {X 0,Y 361.967,Z 742.336,A -85,B 0,C 180,E1 -13208.202,E2 -13208.202} C_VEL
LIN {X 0,Y 362.907,Z 748.042,A -85,B 0,C 180,E1 -13210.19,E2 -13210.19} C_VEL
LIN {X 0,Y 362.917,Z 753.426,A -85,B 0,C 180,E1 -13211.95,E2 -13211.95} C_VEL
LIN {X 0,Y 362.803,Z 755.972,A -85,B 0,C 180,E1 -13212.687,E2 -13212.687} C_VEL
LIN {X 0,Y 363.921,Z 762.022,A -85,B 0,C 180,E1 -13212.914,E2 -13212.914} C_VEL
LIN {X 0,Y 366.732,Z 777.723,A -85,B 0,C 180,E1 -13213.365,E2 -13213.365} C_VEL
LIN {X 0,Y 366.066,Z 831.572,A -85,B 0,C 180,E1 -13214.444,E2 -13214.444} C_VEL
LIN {X 0,Y 365.793,Z 841.389,A -85,B 0,C 180,E1 -13214.789,E2 -13214.789} C_VEL
LIN {X 0,Y 365.22,Z 852.493,A -85,B 0,C 180,E1 -13215.371,E2 -13215.371} C_VEL
LIN {X 0,Y 364.612,Z 863.313,A -85,B 0,C 180,E1 -13216.2,E2 -13216.2} C_VEL
LIN {X 0,Y 363.95,Z 871.703,A -85,B 0,C 180,E1 -13217.028,E2 -13217.028} C_VEL
LIN {X 0,Y 363.329,Z 879.62,A -85,B 0,C 180,E1 -13217.998,E2 -13217.998} C_VEL
LIN {X 0,Y 362.813,Z 885.305,A -85,B 0,C 180,E1 -13218.831,E2 -13218.831} C_VEL
LIN {X 0,Y 362.193,Z 891.652,A -85,B 0,C 180,E1 -13219.943,E2 -13219.943} C_VEL
LIN {X 0,Y 361.599,Z 898.093,A -85,B 0,C 180,E1 -13221.337,E2 -13221.337} C_VEL
LIN {X 0,Y 361.241,Z 903.229,A -85,B 0,C 180,E1 -13222.736,E2 -13222.736} C_VEL
LIN {X 0,Y 360.843,Z 907.98,A -85,B 0,C 180,E1 -13224.411,E2 -13224.411} C_VEL
LIN {X 0,Y 360.613,Z 910.299,A -85,B 0,C 180,E1 -13225.529,E2 -13225.529} C_VEL
LIN {X 0,Y 360.457,Z 912.062,A -85,B 0,C 180,E1 -13226.647,E2 -13226.647} C_VEL
LIN {X 0,Y 360.4,Z 913.331,A -85,B 0,C 180,E1 -13227.765,E2 -13227.765} C_VEL
LIN {X 0,Y 360.354,Z 914.133,A -85,B 0,C 180,E1 -13228.882,E2 -13228.882} C_VEL
LIN {X 0,Y 360.36,Z 914.437,A -85,B 0,C 180,E1 -13230,E2 -13230} C_VEL
LIN {X 0,Y 360.353,Z 914.161,A -85,B 0,C 180,E1 -13231.118,E2 -13231.118} C_VEL
LIN {X 0,Y 360.387,Z 913.417,A -85,B 0,C 180,E1 -13232.235,E2 -13232.235} C_VEL
LIN {X 0,Y 360.455,Z 912.205,A -85,B 0,C 180,E1 -13233.353,E2 -13233.353} C_VEL
LIN {X 0,Y 360.722,Z 909.357,A -85,B 0,C 180,E1 -13235.03,E2 -13235.03} C_VEL
LIN {X 0,Y 360.937,Z 906.765,A -85,B 0,C 180,E1 -13236.148,E2 -13236.148} C_VEL
LIN {X 0,Y 361.179,Z 903.568,A -85,B 0,C 180,E1 -13237.266,E2 -13237.266} C_VEL
LIN {X 0,Y 361.56,Z 898.511,A -85,B 0,C 180,E1 -13238.664,E2 -13238.664} C_VEL
LIN {X 0,Y 362.024,Z 893.567,A -85,B 0,C 180,E1 -13239.78,E2 -13239.78} C_VEL
LIN {X 0,Y 362.627,Z 887.597,A -85,B 0,C 180,E1 -13240.892,E2 -13240.892} C_VEL
LIN {X 0,Y 363.302,Z 880.33,A -85,B 0,C 180,E1 -13242.003,E2 -13242.003} C_VEL
LIN {X 0,Y 363.923,Z 872.563,A -85,B 0,C 180,E1 -13242.973,E2 -13242.973} C_VEL
LIN {X 0,Y 364.46,Z 865.863,A -85,B 0,C 180,E1 -13243.664,E2 -13243.664} C_VEL
LIN {X 0,Y 365.004,Z 857.674,A -85,B 0,C 180,E1 -13244.353,E2 -13244.353} C_VEL
LIN {X 0,Y 365.476,Z 849.372,A -85,B 0,C 180,E1 -13244.904,E2 -13244.904} C_VEL
LIN {X 0,Y 365.831,Z 840.396,A -85,B 0,C 180,E1 -13245.352,E2 -13245.352} C_VEL
LIN {X 0,Y 366.108,Z 830.757,A -85,B 0,C 180,E1 -13245.677,E2 -13245.677} C_VEL
LIN {X 0,Y 366.617,Z 776.304,A -85,B 0,C 180,E1 -13246.769,E2 -13246.769} C_VEL
LIN {X 0,Y 365.646,Z 770.867,A -85,B 0,C 180,E1 -13246.925,E2 -13246.925} C_VEL
LIN {X 0,Y 364.758,Z 767.26,A -85,B 0,C 180,E1 -13247.075,E2 -13247.075} C_VEL
LIN {X 0,Y 362.716,Z 762.385,A -85,B 0,C 180,E1 -13247.444,E2 -13247.444} C_VEL
LIN {X 0,Y 359.538,Z 756.868,A -85,B 0,C 180,E1 -13248.153,E2 -13248.153} C_VEL
LIN {X 0,Y 356.854,Z 752.317,A -85,B 0,C 180,E1 -13249.076,E2 -13249.076} C_VEL
LIN {X 0,Y 355.92,Z 749.527,A -85,B 0,C 180,E1 -13249.886,E2 -13249.886} C_VEL
LIN {X 0,Y 354.908,Z 743.174,A -85,B 0,C 180,E1 -13252.178,E2 -13252.178} C_VEL
LIN {X 0,Y 354.817,Z 743.099,A -85,B 0,C 180,E1 -13255.834,E2 -13255.834} C_VEL
LIN {X 0,Y 354.8,Z 743.102,A -85,B 0,C 180,E1 -13259.684,E2 -13259.684} C_VEL
LIN {X 0,Y 354.788,Z 743.09,A -85,B 0,C 180,E1 -13262.333,E2 -13262.333} C_VEL
LIN {X 0,Y 354.823,Z 743.1,A -85,B 0,C 180,E1 -13265.699,E2 -13265.699} C_VEL
LIN {X 0,Y 354.825,Z 743.081,A -85,B 0,C 180,E1 -13269.424,E2 -13269.424} C_VEL
LIN {X 0,Y 354.789,Z 743.104,A -85,B 0,C 180,E1 -13272.867,E2 -13272.867} C_VEL
LIN {X 0,Y 354.768,Z 743.075,A -85,B 0,C 180,E1 -13276.104,E2 -13276.104} C_VEL
LIN {X 0,Y 354.787,Z 743.073,A -85,B 0,C 180,E1 -13279.179,E2 -13279.179} C_VEL
LIN {X 0,Y 354.808,Z 743.098,A -85,B 0,C 180,E1 -13282.403,E2 -13282.403} C_VEL
LIN {X 0,Y 354.813,Z 743.095,A -85,B 0,C 180,E1 -13284.941,E2 -13284.941} C_VEL
LIN {X 0,Y 354.794,Z 743.095,A -85,B 0,C 180,E1 -13288.405,E2 -13288.405} C_VEL
LIN {X 0,Y 354.848,Z 743.091,A -85,B 0,C 180,E1 -13291.619,E2 -13291.619} C_VEL
LIN {X 0,Y 354.9,Z 743.07,A -85,B 0,C 180,E1 -13294.173,E2 -13294.173} C_VEL
LIN {X 0,Y 354.819,Z 743.097,A -85,B 0,C 180,E1 -13297.893,E2 -13297.893} C_VEL
LIN {X 0,Y 354.853,Z 743.079,A -85,B 0,C 180,E1 -13301.525,E2 -13301.525} C_VEL
LIN {X 0,Y 354.921,Z 743.078,A -85,B 0,C 180,E1 -13305.083,E2 -13305.083} C_VEL
LIN {X 0,Y 354.936,Z 743.082,A -85,B 0,C 180,E1 -13308.579,E2 -13308.579} C_VEL
LIN {X 0,Y 355.115,Z 743.036,A -85,B 0,C 180,E1 -13312.037,E2 -13312.037} C_VEL
LIN {X 0,Y 355.094,Z 743.053,A -85,B 0,C 180,E1 -13314.321,E2 -13314.321} C_VEL
LIN {X 0,Y 355.248,Z 743.045,A -85,B 0,C 180,E1 -13317.732,E2 -13317.732} C_VEL
LIN {X 0,Y 355.398,Z 743.016,A -85,B 0,C 180,E1 -13320,E2 -13320} C_VEL
LIN {X 0,Y 355.245,Z 743.02,A -85,B 0,C 180,E1 -13322.267,E2 -13322.267} C_VEL
LIN {X 0,Y 355.127,Z 743.058,A -85,B 0,C 180,E1 -13326.819,E2 -13326.819} C_VEL
LIN {X 0,Y 354.98,Z 743.067,A -85,B 0,C 180,E1 -13330.264,E2 -13330.264} C_VEL
LIN {X 0,Y 354.944,Z 743.073,A -85,B 0,C 180,E1 -13334.019,E2 -13334.019} C_VEL
LIN {X 0,Y 354.925,Z 743.083,A -85,B 0,C 180,E1 -13338.109,E2 -13338.109} C_VEL
LIN {X 0,Y 354.839,Z 743.081,A -85,B 0,C 180,E1 -13342.106,E2 -13342.106} C_VEL
LIN {X 0,Y 354.9,Z 743.091,A -85,B 0,C 180,E1 -13345.827,E2 -13345.827} C_VEL
LIN {X 0,Y 354.818,Z 743.083,A -85,B 0,C 180,E1 -13349.682,E2 -13349.682} C_VEL
LIN {X 0,Y 354.806,Z 743.101,A -85,B 0,C 180,E1 -13353.702,E2 -13353.702} C_VEL
LIN {X 0,Y 354.802,Z 743.081,A -85,B 0,C 180,E1 -13356.459,E2 -13356.459} C_VEL
LIN {X 0,Y 354.824,Z 743.047,A -85,B 0,C 180,E1 -13359.423,E2 -13359.423} C_VEL
LIN {X 0,Y 354.804,Z 743.095,A -85,B 0,C 180,E1 -13362.87,E2 -13362.87} C_VEL
LIN {X 0,Y 354.768,Z 743.105,A -85,B 0,C 180,E1 -13366.104,E2 -13366.104} C_VEL
LIN {X 0,Y 354.789,Z 743.086,A -85,B 0,C 180,E1 -13369.179,E2 -13369.179} C_VEL
LIN {X 0,Y 354.813,Z 743.101,A -85,B 0,C 180,E1 -13372.401,E2 -13372.401} C_VEL
LIN {X 0,Y 354.813,Z 743.094,A -85,B 0,C 180,E1 -13374.941,E2 -13374.941} C_VEL
LIN {X 0,Y 354.793,Z 743.082,A -85,B 0,C 180,E1 -13378.405,E2 -13378.405} C_VEL
LIN {X 0,Y 354.851,Z 743.097,A -85,B 0,C 180,E1 -13381.619,E2 -13381.619} C_VEL
LIN {X 0,Y 354.921,Z 743.129,A -85,B 0,C 180,E1 -13383.008,E2 -13383.008} C_VEL
LIN {X 0,Y 356.821,Z 753.395,A -85,B 0,C 180,E1 -13386.186,E2 -13386.186} C_VEL
LIN {X 0,Y 357.157,Z 757.42,A -85,B 0,C 180,E1 -13387.351,E2 -13387.351} C_VEL
LIN {X 0,Y 355.817,Z 772.206,A -85,B 0,C 180,E1 -13391.456,E2 -13391.456} C_VEL
LIN {X 0,Y 355.586,Z 775.207,A -85,B 0,C 180,E1 -13392.235,E2 -13392.235} C_VEL
LIN {X 0,Y 356.254,Z 779.612,A -85,B 0,C 180,E1 -13392.422,E2 -13392.422} C_VEL
LIN {X 0,Y 359.648,Z 804.607,A -85,B 0,C 180,E1 -13393.103,E2 -13393.103} C_VEL
LIN {X 0,Y 359.056,Z 852.823,A -85,B 0,C 180,E1 -13394.096,E2 -13394.096} C_VEL
LIN {X 0,Y 358.608,Z 863.227,A -85,B 0,C 180,E1 -13394.476,E2 -13394.476} C_VEL
LIN {X 0,Y 357.984,Z 873.895,A -85,B 0,C 180,E1 -13395.068,E2 -13395.068} C_VEL
LIN {X 0,Y 357.239,Z 884.507,A -85,B 0,C 180,E1 -13395.909,E2 -13395.909} C_VEL
LIN {X 0,Y 356.505,Z 892.822,A -85,B 0,C 180,E1 -13396.752,E2 -13396.752} C_VEL
LIN {X 0,Y 355.776,Z 900.694,A -85,B 0,C 180,E1 -13397.74,E2 -13397.74} C_VEL
LIN {X 0,Y 355.119,Z 908.059,A -85,B 0,C 180,E1 -13398.875,E2 -13398.875} C_VEL
LIN {X 0,Y 354.466,Z 915.532,A -85,B 0,C 180,E1 -13400.298,E2 -13400.298} C_VEL
LIN {X 0,Y 353.849,Z 922.356,A -85,B 0,C 180,E1 -13402.008,E2 -13402.008} C_VEL
LIN {X 0,Y 353.476,Z 927.712,A -85,B 0,C 180,E1 -13403.786,E2 -13403.786} C_VEL
LIN {X 0,Y 353.373,Z 931.354,A -85,B 0,C 180,E1 -13405.437,E2 -13405.437} C_VEL
LIN {X 0,Y 353.248,Z 933.104,A -85,B 0,C 180,E1 -13406.578,E2 -13406.578} C_VEL
LIN {X 0,Y 353.176,Z 934.358,A -85,B 0,C 180,E1 -13407.719,E2 -13407.719} C_VEL
LIN {X 0,Y 353.214,Z 935.14,A -85,B 0,C 180,E1 -13408.86,E2 -13408.86} C_VEL
LIN {X 0,Y 353.26,Z 935.436,A -85,B 0,C 180,E1 -13410,E2 -13410} C_VEL
LIN {X 0,Y 353.214,Z 935.137,A -85,B 0,C 180,E1 -13411.14,E2 -13411.14} C_VEL
LIN {X 0,Y 353.176,Z 934.349,A -85,B 0,C 180,E1 -13412.281,E2 -13412.281} C_VEL
LIN {X 0,Y 353.248,Z 933.089,A -85,B 0,C 180,E1 -13413.422,E2 -13413.422} C_VEL
LIN {X 0,Y 353.365,Z 930.173,A -85,B 0,C 180,E1 -13415.135,E2 -13415.135} C_VEL
LIN {X 0,Y 353.476,Z 927.685,A -85,B 0,C 180,E1 -13416.214,E2 -13416.214} C_VEL
LIN {X 0,Y 353.849,Z 922.32,A -85,B 0,C 180,E1 -13417.992,E2 -13417.992} C_VEL
LIN {X 0,Y 354.455,Z 915.477,A -85,B 0,C 180,E1 -13419.703,E2 -13419.703} C_VEL
LIN {X 0,Y 355.119,Z 908,A -85,B 0,C 180,E1 -13421.125,E2 -13421.125} C_VEL
LIN {X 0,Y 355.775,Z 900.627,A -85,B 0,C 180,E1 -13422.26,E2 -13422.26} C_VEL
LIN {X 0,Y 356.503,Z 892.735,A -85,B 0,C 180,E1 -13423.248,E2 -13423.248} C_VEL
LIN {X 0,Y 357.244,Z 884.397,A -85,B 0,C 180,E1 -13424.09,E2 -13424.09} C_VEL
LIN {X 0,Y 357.963,Z 873.745,A -85,B 0,C 180,E1 -13424.933,E2 -13424.933} C_VEL
LIN {X 0,Y 358.558,Z 862.981,A -85,B 0,C 180,E1 -13425.526,E2 -13425.526} C_VEL
LIN {X 0,Y 359.064,Z 852.435,A -85,B 0,C 180,E1 -13425.904,E2 -13425.904} C_VEL
LIN {X 0,Y 359.544,Z 803.085,A -85,B 0,C 180,E1 -13426.922,E2 -13426.922} C_VEL
LIN {X 0,Y 355.804,Z 777.118,A -85,B 0,C 180,E1 -13427.641,E2 -13427.641} C_VEL
LIN {X 0,Y 355.581,Z 775.214,A -85,B 0,C 180,E1 -13427.758,E2 -13427.758} C_VEL
LIN {X 0,Y 356.739,Z 761.955,A -85,B 0,C 180,E1 -13431.375,E2 -13431.375} C_VEL
LIN {X 0,Y 357.138,Z 755.525,A -85,B 0,C 180,E1 -13433.177,E2 -13433.177} C_VEL
LIN {X 0,Y 355.44,Z 745.884,A -85,B 0,C 180,E1 -13436.075,E2 -13436.075} C_VEL
LIN {X 0,Y 354.921,Z 743.129,A -85,B 0,C 180,E1 -13436.992,E2 -13436.992} C_VEL
LIN {X 0,Y 354.854,Z 743.077,A -85,B 0,C 180,E1 -13439.679,E2 -13439.679} C_VEL
LIN {X 0,Y 354.806,Z 743.104,A -85,B 0,C 180,E1 -13443.702,E2 -13443.702} C_VEL
LIN {X 0,Y 354.802,Z 743.093,A -85,B 0,C 180,E1 -13446.459,E2 -13446.459} C_VEL
LIN {X 0,Y 354.824,Z 743.093,A -85,B 0,C 180,E1 -13449.424,E2 -13449.424} C_VEL
LIN {X 0,Y 354.788,Z 743.092,A -85,B 0,C 180,E1 -13452.867,E2 -13452.867} C_VEL
LIN {X 0,Y 354.776,Z 743.101,A -85,B 0,C 180,E1 -13456.105,E2 -13456.105} C_VEL
LIN {X 0,Y 354.825,Z 743.06,A -85,B 0,C 180,E1 -13459.184,E2 -13459.184} C_VEL
LIN {X 0,Y 354.814,Z 743.069,A -85,B 0,C 180,E1 -13462.401,E2 -13462.401} C_VEL
LIN {X 0,Y 354.813,Z 743.093,A -85,B 0,C 180,E1 -13464.941,E2 -13464.941} C_VEL
LIN {X 0,Y 354.794,Z 743.096,A -85,B 0,C 180,E1 -13468.405,E2 -13468.405} C_VEL
LIN {X 0,Y 354.847,Z 743.083,A -85,B 0,C 180,E1 -13471.619,E2 -13471.619} C_VEL
LIN {X 0,Y 354.9,Z 743.091,A -85,B 0,C 180,E1 -13474.173,E2 -13474.173} C_VEL
LIN {X 0,Y 354.839,Z 743.081,A -85,B 0,C 180,E1 -13477.894,E2 -13477.894} C_VEL
LIN {X 0,Y 354.925,Z 743.083,A -85,B 0,C 180,E1 -13481.891,E2 -13481.891} C_VEL
LIN {X 0,Y 354.944,Z 743.072,A -85,B 0,C 180,E1 -13485.981,E2 -13485.981} C_VEL
LIN {X 0,Y 354.98,Z 743.067,A -85,B 0,C 180,E1 -13489.736,E2 -13489.736} C_VEL
LIN {X 0,Y 355.127,Z 743.058,A -85,B 0,C 180,E1 -13493.181,E2 -13493.181} C_VEL
LIN {X 0,Y 355.246,Z 743.019,A -85,B 0,C 180,E1 -13497.733,E2 -13497.733} C_VEL
LIN {X 0,Y 355.4,Z 743.015,A -85,B 0,C 180,E1 -13500,E2 -13500} C_VEL
LIN {X 0,Y 355.248,Z 743.045,A -85,B 0,C 180,E1 -13502.268,E2 -13502.268} C_VEL
LIN {X 0,Y 355.139,Z 743.036,A -85,B 0,C 180,E1 -13506.819,E2 -13506.819} C_VEL
LIN {X 0,Y 355.017,Z 743.061,A -85,B 0,C 180,E1 -13509.112,E2 -13509.112} C_VEL
LIN {X 0,Y 354.923,Z 743.088,A -85,B 0,C 180,E1 -13512.581,E2 -13512.581} C_VEL
LIN {X 0,Y 354.888,Z 743.077,A -85,B 0,C 180,E1 -13516.096,E2 -13516.096} C_VEL
LIN {X 0,Y 354.856,Z 743.089,A -85,B 0,C 180,E1 -13519.675,E2 -13519.675} C_VEL
LIN {X 0,Y 354.827,Z 743.093,A -85,B 0,C 180,E1 -13523.337,E2 -13523.337} C_VEL
LIN {X 0,Y 354.889,Z 743.076,A -85,B 0,C 180,E1 -13526.981,E2 -13526.981} C_VEL
LIN {X 0,Y 354.819,Z 743.098,A -85,B 0,C 180,E1 -13529.682,E2 -13529.682} C_VEL
LIN {X 0,Y 354.807,Z 743.089,A -85,B 0,C 180,E1 -13533.702,E2 -13533.702} C_VEL
LIN {X 0,Y 354.798,Z 743.1,A -85,B 0,C 180,E1 -13536.46,E2 -13536.46} C_VEL
LIN {X 0,Y 354.825,Z 743.086,A -85,B 0,C 180,E1 -13539.424,E2 -13539.424} C_VEL
LIN {X 0,Y 354.788,Z 743.056,A -85,B 0,C 180,E1 -13542.867,E2 -13542.867} C_VEL
LIN {X 0,Y 354.768,Z 743.103,A -85,B 0,C 180,E1 -13546.104,E2 -13546.104} C_VEL
LIN {X 0,Y 354.789,Z 743.1,A -85,B 0,C 180,E1 -13549.179,E2 -13549.179} C_VEL
LIN {X 0,Y 354.808,Z 743.082,A -85,B 0,C 180,E1 -13552.403,E2 -13552.403} C_VEL
LIN {X 0,Y 354.813,Z 743.102,A -85,B 0,C 180,E1 -13554.941,E2 -13554.941} C_VEL
LIN {X 0,Y 354.794,Z 743.088,A -85,B 0,C 180,E1 -13558.405,E2 -13558.405} C_VEL
LIN {X 0,Y 354.803,Z 743.101,A -85,B 0,C 180,E1 -13561.615,E2 -13561.615} C_VEL
LIN {X 0,Y 354.852,Z 743.098,A -85,B 0,C 180,E1 -13565.423,E2 -13565.423} C_VEL
LIN {X 0,Y 354.895,Z 743.22,A -85,B 0,C 180,E1 -13567.986,E2 -13567.986} C_VEL
LIN {X 0,Y 355.977,Z 750.03,A -85,B 0,C 180,E1 -13570.389,E2 -13570.389} C_VEL
LIN {X 0,Y 355.848,Z 756.037,A -85,B 0,C 180,E1 -13572.317,E2 -13572.317} C_VEL
LIN {X 0,Y 356.283,Z 758.458,A -85,B 0,C 180,E1 -13572.456,E2 -13572.456} C_VEL
LIN {X 0,Y 359.943,Z 778.127,A -85,B 0,C 180,E1 -13573.046,E2 -13573.046} C_VEL
LIN {X 0,Y 359.24,Z 831.799,A -85,B 0,C 180,E1 -13574.141,E2 -13574.141} C_VEL
LIN {X 0,Y 359.018,Z 840.778,A -85,B 0,C 180,E1 -13574.458,E2 -13574.458} C_VEL
LIN {X 0,Y 358.511,Z 850.314,A -85,B 0,C 180,E1 -13574.945,E2 -13574.945} C_VEL
LIN {X 0,Y 357.962,Z 860.315,A -85,B 0,C 180,E1 -13575.648,E2 -13575.648} C_VEL
LIN {X 0,Y 357.095,Z 870.691,A -85,B 0,C 180,E1 -13576.629,E2 -13576.629} C_VEL
LIN {X 0,Y 356.474,Z 878.815,A -85,B 0,C 180,E1 -13577.619,E2 -13577.619} C_VEL
LIN {X 0,Y 355.861,Z 885.517,A -85,B 0,C 180,E1 -13578.61,E2 -13578.61} C_VEL
LIN {X 0,Y 355.218,Z 891.863,A -85,B 0,C 180,E1 -13579.743,E2 -13579.743} C_VEL
LIN {X 0,Y 354.599,Z 898.303,A -85,B 0,C 180,E1 -13581.164,E2 -13581.164} C_VEL
LIN {X 0,Y 354.202,Z 903.44,A -85,B 0,C 180,E1 -13582.59,E2 -13582.59} C_VEL
LIN {X 0,Y 353.781,Z 908.19,A -85,B 0,C 180,E1 -13584.3,E2 -13584.3} C_VEL
LIN {X 0,Y 353.555,Z 910.508,A -85,B 0,C 180,E1 -13585.439,E2 -13585.439} C_VEL
LIN {X 0,Y 353.377,Z 912.271,A -85,B 0,C 180,E1 -13586.579,E2 -13586.579} C_VEL
LIN {X 0,Y 353.305,Z 913.54,A -85,B 0,C 180,E1 -13587.72,E2 -13587.72} C_VEL
LIN {X 0,Y 353.258,Z 914.342,A -85,B 0,C 180,E1 -13588.86,E2 -13588.86} C_VEL
LIN {X 0,Y 353.264,Z 914.646,A -85,B 0,C 180,E1 -13590,E2 -13590} C_VEL
LIN {X 0,Y 353.257,Z 914.37,A -85,B 0,C 180,E1 -13591.14,E2 -13591.14} C_VEL
LIN {X 0,Y 353.292,Z 913.625,A -85,B 0,C 180,E1 -13592.28,E2 -13592.28} C_VEL
LIN {X 0,Y 353.376,Z 912.413,A -85,B 0,C 180,E1 -13593.421,E2 -13593.421} C_VEL
LIN {X 0,Y 353.67,Z 909.564,A -85,B 0,C 180,E1 -13595.13,E2 -13595.13} C_VEL
LIN {X 0,Y 353.903,Z 906.414,A -85,B 0,C 180,E1 -13596.483,E2 -13596.483} C_VEL
LIN {X 0,Y 354.263,Z 901.873,A -85,B 0,C 180,E1 -13597.982,E2 -13597.982} C_VEL
LIN {X 0,Y 354.755,Z 896.383,A -85,B 0,C 180,E1 -13599.407,E2 -13599.407} C_VEL
LIN {X 0,Y 355.513,Z 889.48,A -85,B 0,C 180,E1 -13600.825,E2 -13600.825} C_VEL
LIN {X 0,Y 356.299,Z 881.552,A -85,B 0,C 180,E1 -13602.098,E2 -13602.098} C_VEL
LIN {X 0,Y 356.939,Z 873.993,A -85,B 0,C 180,E1 -13603.087,E2 -13603.087} C_VEL
LIN {X 0,Y 357.459,Z 867.564,A -85,B 0,C 180,E1 -13603.792,E2 -13603.792} C_VEL
LIN {X 0,Y 358.007,Z 859.746,A -85,B 0,C 180,E1 -13604.495,E2 -13604.495} C_VEL
LIN {X 0,Y 358.592,Z 850.779,A -85,B 0,C 180,E1 -13605.124,E2 -13605.124} C_VEL
LIN {X 0,Y 358.975,Z 841.423,A -85,B 0,C 180,E1 -13605.617,E2 -13605.617} C_VEL
LIN {X 0,Y 359.221,Z 832.083,A -85,B 0,C 180,E1 -13605.953,E2 -13605.953} C_VEL
LIN {X 0,Y 359.897,Z 777.576,A -85,B 0,C 180,E1 -13607.069,E2 -13607.069} C_VEL
LIN {X 0,Y 355.837,Z 756.004,A -85,B 0,C 180,E1 -13607.744,E2 -13607.744} C_VEL
LIN {X 0,Y 356.001,Z 750.337,A -85,B 0,C 180,E1 -13609.609,E2 -13609.609} C_VEL
LIN {X 0,Y 355.92,Z 749.527,A -85,B 0,C 180,E1 -13609.886,E2 -13609.886} C_VEL
LIN {X 0,Y 355.038,Z 748.006,A -85,B 0,C 180,E1 -13610.457,E2 -13610.457} C_VEL
LIN {X 0,Y 351.802,Z 746.02,A -85,B 0,C 180,E1 -13611.361,E2 -13611.361} C_VEL
LIN {X 0,Y 348.603,Z 744.378,A -85,B 0,C 180,E1 -13612.312,E2 -13612.312} C_VEL
LIN {X 0,Y 347.807,Z 743.979,A -85,B 0,C 180,E1 -13612.954,E2 -13612.954} C_VEL
LIN {X 0,Y 347.752,Z 743.981,A -85,B 0,C 180,E1 -13616.399,E2 -13616.399} C_VEL
LIN {X 0,Y 347.742,Z 743.976,A -85,B 0,C 180,E1 -13620.349,E2 -13620.349} C_VEL
LIN {X 0,Y 347.749,Z 743.98,A -85,B 0,C 180,E1 -13624.044,E2 -13624.044} C_VEL
LIN {X 0,Y 347.762,Z 743.964,A -85,B 0,C 180,E1 -13627.321,E2 -13627.321} C_VEL
LIN {X 0,Y 347.733,Z 743.969,A -85,B 0,C 180,E1 -13630.297,E2 -13630.297} C_VEL
LIN {X 0,Y 347.724,Z 743.98,A -85,B 0,C 180,E1 -13633.408,E2 -13633.408} C_VEL
LIN {X 0,Y 347.726,Z 743.941,A -85,B 0,C 180,E1 -13636.686,E2 -13636.686} C_VEL
LIN {X 0,Y 347.748,Z 743.962,A -85,B 0,C 180,E1 -13640.173,E2 -13640.173} C_VEL
LIN {X 0,Y 347.763,Z 743.979,A -85,B 0,C 180,E1 -13642.679,E2 -13642.679} C_VEL
LIN {X 0,Y 347.749,Z 743.969,A -85,B 0,C 180,E1 -13645.956,E2 -13645.956} C_VEL
LIN {X 0,Y 347.75,Z 743.978,A -85,B 0,C 180,E1 -13649.652,E2 -13649.652} C_VEL
LIN {X 0,Y 347.832,Z 743.951,A -85,B 0,C 180,E1 -13653.608,E2 -13653.608} C_VEL
LIN {X 0,Y 347.787,Z 743.967,A -85,B 0,C 180,E1 -13656.162,E2 -13656.162} C_VEL
LIN {X 0,Y 347.81,Z 743.967,A -85,B 0,C 180,E1 -13659.909,E2 -13659.909} C_VEL
LIN {X 0,Y 347.834,Z 743.952,A -85,B 0,C 180,E1 -13663.568,E2 -13663.568} C_VEL
LIN {X 0,Y 347.892,Z 743.963,A -85,B 0,C 180,E1 -13667.16,E2 -13667.16} C_VEL
LIN {X 0,Y 348.096,Z 743.913,A -85,B 0,C 180,E1 -13671.612,E2 -13671.612} C_VEL
LIN {X 0,Y 348.069,Z 743.928,A -85,B 0,C 180,E1 -13674.206,E2 -13674.206} C_VEL
LIN {X 0,Y 348.21,Z 743.922,A -85,B 0,C 180,E1 -13677.686,E2 -13677.686} C_VEL
LIN {X 0,Y 348.346,Z 743.894,A -85,B 0,C 180,E1 -13680,E2 -13680} C_VEL
LIN {X 0,Y 348.208,Z 743.896,A -85,B 0,C 180,E1 -13682.313,E2 -13682.313} C_VEL
LIN {X 0,Y 348.092,Z 743.935,A -85,B 0,C 180,E1 -13686.958,E2 -13686.958} C_VEL
LIN {X 0,Y 347.93,Z 743.943,A -85,B 0,C 180,E1 -13690.474,E2 -13690.474} C_VEL
LIN {X 0,Y 347.9,Z 743.952,A -85,B 0,C 180,E1 -13694.15,E2 -13694.15} C_VEL
LIN {X 0,Y 347.893,Z 743.957,A -85,B 0,C 180,E1 -13698.291,E2 -13698.291} C_VEL
LIN {X 0,Y 347.797,Z 743.954,A -85,B 0,C 180,E1 -13701.638,E2 -13701.638} C_VEL
LIN {X 0,Y 347.813,Z 743.969,A -85,B 0,C 180,E1 -13705.108,E2 -13705.108} C_VEL
LIN {X 0,Y 347.809,Z 743.968,A -85,B 0,C 180,E1 -13707.694,E2 -13707.694} C_VEL
LIN {X 0,Y 347.75,Z 743.969,A -85,B 0,C 180,E1 -13710.348,E2 -13710.348} C_VEL
LIN {X 0,Y 347.749,Z 743.981,A -85,B 0,C 180,E1 -13714.044,E2 -13714.044} C_VEL
LIN {X 0,Y 347.767,Z 743.951,A -85,B 0,C 180,E1 -13717.32,E2 -13717.32} C_VEL
LIN {X 0,Y 347.755,Z 743.933,A -85,B 0,C 180,E1 -13720.294,E2 -13720.294} C_VEL
LIN {X 0,Y 347.744,Z 743.975,A -85,B 0,C 180,E1 -13723.405,E2 -13723.405} C_VEL
LIN {X 0,Y 347.725,Z 743.974,A -85,B 0,C 180,E1 -13726.686,E2 -13726.686} C_VEL
LIN {X 0,Y 347.747,Z 743.971,A -85,B 0,C 180,E1 -13730.173,E2 -13730.173} C_VEL
LIN {X 0,Y 347.766,Z 743.974,A -85,B 0,C 180,E1 -13732.68,E2 -13732.68} C_VEL
LIN {X 0,Y 347.748,Z 743.98,A -85,B 0,C 180,E1 -13735.956,E2 -13735.956} C_VEL
LIN {X 0,Y 347.764,Z 743.952,A -85,B 0,C 180,E1 -13739.653,E2 -13739.653} C_VEL
LIN {X 0,Y 347.855,Z 744.024,A -85,B 0,C 180,E1 -13742.744,E2 -13742.744} C_VEL
LIN {X 0,Y 349.768,Z 754.292,A -85,B 0,C 180,E1 -13745.99,E2 -13745.99} C_VEL
LIN {X 0,Y 350.188,Z 757.531,A -85,B 0,C 180,E1 -13746.962,E2 -13746.962} C_VEL
LIN {X 0,Y 349.199,Z 768.174,A -85,B 0,C 180,E1 -13749.992,E2 -13749.992} C_VEL
LIN {X 0,Y 348.631,Z 774.967,A -85,B 0,C 180,E1 -13751.863,E2 -13751.863} C_VEL
LIN {X 0,Y 349.144,Z 778.544,A -85,B 0,C 180,E1 -13752.034,E2 -13752.034} C_VEL
LIN {X 0,Y 352.791,Z 804.008,A -85,B 0,C 180,E1 -13752.755,E2 -13752.755} C_VEL
LIN {X 0,Y 352.269,Z 851.846,A -85,B 0,C 180,E1 -13753.759,E2 -13753.759} C_VEL
LIN {X 0,Y 351.83,Z 861.363,A -85,B 0,C 180,E1 -13754.095,E2 -13754.095} C_VEL
LIN {X 0,Y 351.277,Z 871.398,A -85,B 0,C 180,E1 -13754.628,E2 -13754.628} C_VEL
LIN {X 0,Y 350.48,Z 882.799,A -85,B 0,C 180,E1 -13755.484,E2 -13755.484} C_VEL
LIN {X 0,Y 349.751,Z 891.386,A -85,B 0,C 180,E1 -13756.343,E2 -13756.343} C_VEL
LIN {X 0,Y 348.946,Z 899.465,A -85,B 0,C 180,E1 -13757.348,E2 -13757.348} C_VEL
LIN {X 0,Y 348.324,Z 906.143,A -85,B 0,C 180,E1 -13758.36,E2 -13758.36} C_VEL
LIN {X 0,Y 347.696,Z 912.483,A -85,B 0,C 180,E1 -13759.519,E2 -13759.519} C_VEL
LIN {X 0,Y 347.208,Z 917.753,A -85,B 0,C 180,E1 -13760.681,E2 -13760.681} C_VEL
LIN {X 0,Y 346.803,Z 922.148,A -85,B 0,C 180,E1 -13761.845,E2 -13761.845} C_VEL
LIN {X 0,Y 346.424,Z 927.336,A -85,B 0,C 180,E1 -13763.594,E2 -13763.594} C_VEL
LIN {X 0,Y 346.285,Z 931.145,A -85,B 0,C 180,E1 -13765.344,E2 -13765.344} C_VEL
LIN {X 0,Y 346.175,Z 932.896,A -85,B 0,C 180,E1 -13766.508,E2 -13766.508} C_VEL
LIN {X 0,Y 346.088,Z 934.149,A -85,B 0,C 180,E1 -13767.672,E2 -13767.672} C_VEL
LIN {X 0,Y 346.114,Z 934.931,A -85,B 0,C 180,E1 -13768.837,E2 -13768.837} C_VEL
LIN {X 0,Y 346.163,Z 935.228,A -85,B 0,C 180,E1 -13770,E2 -13770} C_VEL
LIN {X 0,Y 346.114,Z 934.928,A -85,B 0,C 180,E1 -13771.163,E2 -13771.163} C_VEL
LIN {X 0,Y 346.088,Z 934.14,A -85,B 0,C 180,E1 -13772.328,E2 -13772.328} C_VEL
LIN {X 0,Y 346.175,Z 932.88,A -85,B 0,C 180,E1 -13773.492,E2 -13773.492} C_VEL
LIN {X 0,Y 346.269,Z 929.963,A -85,B 0,C 180,E1 -13775.24,E2 -13775.24} C_VEL
LIN {X 0,Y 346.469,Z 926.808,A -85,B 0,C 180,E1 -13776.596,E2 -13776.596} C_VEL
LIN {X 0,Y 346.884,Z 921.146,A -85,B 0,C 180,E1 -13778.447,E2 -13778.447} C_VEL
LIN {X 0,Y 347.447,Z 915.266,A -85,B 0,C 180,E1 -13779.9,E2 -13779.9} C_VEL
LIN {X 0,Y 348.15,Z 907.788,A -85,B 0,C 180,E1 -13781.351,E2 -13781.351} C_VEL
LIN {X 0,Y 348.833,Z 900.415,A -85,B 0,C 180,E1 -13782.508,E2 -13782.508} C_VEL
LIN {X 0,Y 349.605,Z 892.523,A -85,B 0,C 180,E1 -13783.515,E2 -13783.515} C_VEL
LIN {X 0,Y 350.355,Z 884.184,A -85,B 0,C 180,E1 -13784.373,E2 -13784.373} C_VEL
LIN {X 0,Y 351.126,Z 873.531,A -85,B 0,C 180,E1 -13785.231,E2 -13785.231} C_VEL
LIN {X 0,Y 351.731,Z 862.763,A -85,B 0,C 180,E1 -13785.835,E2 -13785.835} C_VEL
LIN {X 0,Y 352.249,Z 852.212,A -85,B 0,C 180,E1 -13786.22,E2 -13786.22} C_VEL
LIN {X 0,Y 352.752,Z 803.719,A -85,B 0,C 180,E1 -13787.24,E2 -13787.24} C_VEL
LIN {X 0,Y 348.991,Z 777.707,A -85,B 0,C 180,E1 -13787.979,E2 -13787.979} C_VEL
LIN {X 0,Y 348.632,Z 775.194,A -85,B 0,C 180,E1 -13788.094,E2 -13788.094} C_VEL
LIN {X 0,Y 349.292,Z 767.076,A -85,B 0,C 180,E1 -13790.309,E2 -13790.309} C_VEL
LIN {X 0,Y 350.179,Z 757.484,A -85,B 0,C 180,E1 -13793.039,E2 -13793.039} C_VEL
LIN {X 0,Y 349.169,Z 750.764,A -85,B 0,C 180,E1 -13795.076,E2 -13795.076} C_VEL
LIN {X 0,Y 347.855,Z 744.017,A -85,B 0,C 180,E1 -13797.256,E2 -13797.256} C_VEL
LIN {X 0,Y 347.764,Z 743.953,A -85,B 0,C 180,E1 -13800.347,E2 -13800.347} C_VEL
LIN {X 0,Y 347.745,Z 743.981,A -85,B 0,C 180,E1 -13804.464,E2 -13804.464} C_VEL
LIN {X 0,Y 347.778,Z 743.977,A -85,B 0,C 180,E1 -13807.99,E2 -13807.99} C_VEL
LIN {X 0,Y 347.751,Z 743.962,A -85,B 0,C 180,E1 -13811.83,E2 -13811.83} C_VEL
LIN {X 0,Y 347.737,Z 743.981,A -85,B 0,C 180,E1 -13815.022,E2 -13815.022} C_VEL
LIN {X 0,Y 347.768,Z 743.954,A -85,B 0,C 180,E1 -13818.394,E2 -13818.394} C_VEL
LIN {X 0,Y 347.779,Z 743.935,A -85,B 0,C 180,E1 -13822.01,E2 -13822.01} C_VEL
LIN {X 0,Y 347.745,Z 743.977,A -85,B 0,C 180,E1 -13825.536,E2 -13825.536} C_VEL
LIN {X 0,Y 347.746,Z 743.975,A -85,B 0,C 180,E1 -13828.301,E2 -13828.301} C_VEL
LIN {X 0,Y 347.779,Z 743.96,A -85,B 0,C 180,E1 -13830.988,E2 -13830.988} C_VEL
LIN {X 0,Y 347.832,Z 743.968,A -85,B 0,C 180,E1 -13833.608,E2 -13833.608} C_VEL
LIN {X 0,Y 347.79,Z 743.969,A -85,B 0,C 180,E1 -13836.162,E2 -13836.162} C_VEL
LIN {X 0,Y 347.829,Z 743.955,A -85,B 0,C 180,E1 -13839.91,E2 -13839.91} C_VEL
LIN {X 0,Y 347.868,Z 743.967,A -85,B 0,C 180,E1 -13842.36,E2 -13842.36} C_VEL
LIN {X 0,Y 347.899,Z 743.949,A -85,B 0,C 180,E1 -13845.971,E2 -13845.971} C_VEL
LIN {X 0,Y 347.93,Z 743.944,A -85,B 0,C 180,E1 -13849.526,E2 -13849.526} C_VEL
LIN {X 0,Y 348.093,Z 743.935,A -85,B 0,C 180,E1 -13853.042,E2 -13853.042} C_VEL
LIN {X 0,Y 348.208,Z 743.895,A -85,B 0,C 180,E1 -13857.687,E2 -13857.687} C_VEL
LIN {X 0,Y 348.348,Z 743.894,A -85,B 0,C 180,E1 -13860,E2 -13860} C_VEL
LIN {X 0,Y 348.21,Z 743.922,A -85,B 0,C 180,E1 -13862.314,E2 -13862.314} C_VEL
LIN {X 0,Y 348.107,Z 743.91,A -85,B 0,C 180,E1 -13866.958,E2 -13866.958} C_VEL
LIN {X 0,Y 347.969,Z 743.942,A -85,B 0,C 180,E1 -13869.299,E2 -13869.299} C_VEL
LIN {X 0,Y 347.892,Z 743.964,A -85,B 0,C 180,E1 -13872.84,E2 -13872.84} C_VEL
LIN {X 0,Y 347.834,Z 743.952,A -85,B 0,C 180,E1 -13876.432,E2 -13876.432} C_VEL
LIN {X 0,Y 347.807,Z 743.967,A -85,B 0,C 180,E1 -13880.091,E2 -13880.091} C_VEL
LIN {X 0,Y 347.786,Z 743.967,A -85,B 0,C 180,E1 -13883.838,E2 -13883.838} C_VEL
LIN {X 0,Y 347.851,Z 743.956,A -85,B 0,C 180,E1 -13887.255,E2 -13887.255} C_VEL
LIN {X 0,Y 347.751,Z 743.978,A -85,B 0,C 180,E1 -13890.348,E2 -13890.348} C_VEL
LIN {X 0,Y 347.749,Z 743.969,A -85,B 0,C 180,E1 -13894.044,E2 -13894.044} C_VEL
LIN {X 0,Y 347.763,Z 743.98,A -85,B 0,C 180,E1 -13897.321,E2 -13897.321} C_VEL
LIN {X 0,Y 347.733,Z 743.963,A -85,B 0,C 180,E1 -13900.297,E2 -13900.297} C_VEL
LIN {X 0,Y 347.724,Z 743.94,A -85,B 0,C 180,E1 -13903.408,E2 -13903.408} C_VEL
LIN {X 0,Y 347.726,Z 743.98,A -85,B 0,C 180,E1 -13906.686,E2 -13906.686} C_VEL
LIN {X 0,Y 347.748,Z 743.965,A -85,B 0,C 180,E1 -13910.173,E2 -13910.173} C_VEL
LIN {X 0,Y 347.762,Z 743.962,A -85,B 0,C 180,E1 -13912.679,E2 -13912.679} C_VEL
LIN {X 0,Y 347.749,Z 743.981,A -85,B 0,C 180,E1 -13915.956,E2 -13915.956} C_VEL
LIN {X 0,Y 347.742,Z 743.974,A -85,B 0,C 180,E1 -13919.651,E2 -13919.651} C_VEL
LIN {X 0,Y 347.757,Z 743.982,A -85,B 0,C 180,E1 -13923.602,E2 -13923.602} C_VEL
LIN {X 0,Y 347.774,Z 743.971,A -85,B 0,C 180,E1 -13926.161,E2 -13926.161} C_VEL
LIN {X 0,Y 347.855,Z 744.154,A -85,B 0,C 180,E1 -13927.787,E2 -13927.787} C_VEL
LIN {X 0,Y 348.89,Z 750.227,A -85,B 0,C 180,E1 -13929.974,E2 -13929.974} C_VEL
LIN {X 0,Y 348.923,Z 755.966,A -85,B 0,C 180,E1 -13931.891,E2 -13931.891} C_VEL
LIN {X 0,Y 349.042,Z 757.276,A -85,B 0,C 180,E1 -13932.04,E2 -13932.04} C_VEL
LIN {X 0,Y 353.098,Z 778.463,A -85,B 0,C 180,E1 -13932.709,E2 -13932.709} C_VEL
LIN {X 0,Y 352.435,Z 832.026,A -85,B 0,C 180,E1 -13933.826,E2 -13933.826} C_VEL
LIN {X 0,Y 352.198,Z 840.998,A -85,B 0,C 180,E1 -13934.149,E2 -13934.149} C_VEL
LIN {X 0,Y 351.689,Z 850.53,A -85,B 0,C 180,E1 -13934.646,E2 -13934.646} C_VEL
LIN {X 0,Y 351.113,Z 860.53,A -85,B 0,C 180,E1 -13935.362,E2 -13935.362} C_VEL
LIN {X 0,Y 350.215,Z 870.903,A -85,B 0,C 180,E1 -13936.361,E2 -13936.361} C_VEL
LIN {X 0,Y 349.559,Z 879.027,A -85,B 0,C 180,E1 -13937.371,E2 -13937.371} C_VEL
LIN {X 0,Y 348.917,Z 885.728,A -85,B 0,C 180,E1 -13938.38,E2 -13938.38} C_VEL
LIN {X 0,Y 348.255,Z 892.073,A -85,B 0,C 180,E1 -13939.536,E2 -13939.536} C_VEL
LIN {X 0,Y 347.704,Z 897.346,A -85,B 0,C 180,E1 -13940.694,E2 -13940.694} C_VEL
LIN {X 0,Y 347.299,Z 901.746,A -85,B 0,C 180,E1 -13941.856,E2 -13941.856} C_VEL
LIN {X 0,Y 346.984,Z 905.409,A -85,B 0,C 180,E1 -13943.02,E2 -13943.02} C_VEL
LIN {X 0,Y 346.725,Z 908.4,A -85,B 0,C 180,E1 -13944.183,E2 -13944.183} C_VEL
LIN {X 0,Y 346.5,Z 910.717,A -85,B 0,C 180,E1 -13945.346,E2 -13945.346} C_VEL
LIN {X 0,Y 346.301,Z 912.48,A -85,B 0,C 180,E1 -13946.509,E2 -13946.509} C_VEL
LIN {X 0,Y 346.212,Z 913.75,A -85,B 0,C 180,E1 -13947.673,E2 -13947.673} C_VEL
LIN {X 0,Y 346.162,Z 914.551,A -85,B 0,C 180,E1 -13948.837,E2 -13948.837} C_VEL
LIN {X 0,Y 346.167,Z 914.855,A -85,B 0,C 180,E1 -13950,E2 -13950} C_VEL
LIN {X 0,Y 346.16,Z 914.579,A -85,B 0,C 180,E1 -13951.163,E2 -13951.163} C_VEL
LIN {X 0,Y 346.2,Z 913.834,A -85,B 0,C 180,E1 -13952.327,E2 -13952.327} C_VEL
LIN {X 0,Y 346.3,Z 912.621,A -85,B 0,C 180,E1 -13953.491,E2 -13953.491} C_VEL
LIN {X 0,Y 346.619,Z 909.772,A -85,B 0,C 180,E1 -13955.235,E2 -13955.235} C_VEL
LIN {X 0,Y 346.81,Z 907.042,A -85,B 0,C 180,E1 -13956.453,E2 -13956.453} C_VEL
LIN {X 0,Y 347.225,Z 902.081,A -85,B 0,C 180,E1 -13958.145,E2 -13958.145} C_VEL
LIN {X 0,Y 347.764,Z 896.59,A -85,B 0,C 180,E1 -13959.597,E2 -13959.597} C_VEL
LIN {X 0,Y 348.555,Z 889.686,A -85,B 0,C 180,E1 -13961.043,E2 -13961.043} C_VEL
LIN {X 0,Y 349.358,Z 881.758,A -85,B 0,C 180,E1 -13962.342,E2 -13962.342} C_VEL
LIN {X 0,Y 350.042,Z 874.197,A -85,B 0,C 180,E1 -13963.35,E2 -13963.35} C_VEL
LIN {X 0,Y 350.593,Z 867.766,A -85,B 0,C 180,E1 -13964.067,E2 -13964.067} C_VEL
LIN {X 0,Y 351.159,Z 859.948,A -85,B 0,C 180,E1 -13964.784,E2 -13964.784} C_VEL
LIN {X 0,Y 351.763,Z 850.979,A -85,B 0,C 180,E1 -13965.425,E2 -13965.425} C_VEL
LIN {X 0,Y 352.159,Z 841.62,A -85,B 0,C 180,E1 -13965.927,E2 -13965.927} C_VEL
LIN {X 0,Y 352.407,Z 832.362,A -85,B 0,C 180,E1 -13966.268,E2 -13966.268} C_VEL
LIN {X 0,Y 353.11,Z 778.625,A -85,B 0,C 180,E1 -13967.39,E2 -13967.39} C_VEL
LIN {X 0,Y 348.883,Z 756.326,A -85,B 0,C 180,E1 -13968.082,E2 -13968.082} C_VEL
LIN {X 0,Y 348.918,Z 750.538,A -85,B 0,C 180,E1 -13970.024,E2 -13970.024} C_VEL
LIN {X 0,Y 347.86,Z 744.058,A -85,B 0,C 180,E1 -13972.398,E2 -13972.398} C_VEL
LIN {X 0,Y 347.807,Z 743.979,A -85,B 0,C 180,E1 -13972.954,E2 -13972.954} C_VEL
LIN {X 0,Y 347.086,Z 744.06,A -85,B 0,C 180,E1 -13973.92,E2 -13973.92} C_VEL
LIN {X 0,Y 344.2,Z 744.423,A -85,B 0,C 180,E1 -13975.49,E2 -13975.49} C_VEL
LIN {X 0,Y 341.789,Z 744.724,A -85,B 0,C 180,E1 -13976.761,E2 -13976.761} C_VEL
LIN {X 0,Y 340.763,Z 744.849,A -85,B 0,C 180,E1 -13977.745,E2 -13977.745} C_VEL
LIN {X 0,Y 340.682,Z 744.858,A -85,B 0,C 180,E1 -13978.078,E2 -13978.078} C_VEL
LIN {X 0,Y 340.695,Z 744.847,A -85,B 0,C 180,E1 -13981.045,E2 -13981.045} C_VEL
LIN {X 0,Y 340.719,Z 744.857,A -85,B 0,C 180,E1 -13985.279,E2 -13985.279} C_VEL
LIN {X 0,Y 340.71,Z 744.832,A -85,B 0,C 180,E1 -13988.386,E2 -13988.386} C_VEL
LIN {X 0,Y 340.7,Z 744.857,A -85,B 0,C 180,E1 -13992.045,E2 -13992.045} C_VEL
LIN {X 0,Y 340.653,Z 744.828,A -85,B 0,C 180,E1 -13996.227,E2 -13996.227} C_VEL
LIN {X 0,Y 340.689,Z 744.839,A -85,B 0,C 180,E1 -13999.753,E2 -13999.753} C_VEL
LIN {X 0,Y 340.706,Z 744.857,A -85,B 0,C 180,E1 -14003.258,E2 -14003.258} C_VEL
LIN {X 0,Y 340.693,Z 744.848,A -85,B 0,C 180,E1 -14006.153,E2 -14006.153} C_VEL
LIN {X 0,Y 340.743,Z 744.852,A -85,B 0,C 180,E1 -14010.329,E2 -14010.329} C_VEL
LIN {X 0,Y 340.804,Z 744.831,A -85,B 0,C 180,E1 -14013.02,E2 -14013.02} C_VEL
LIN {X 0,Y 340.756,Z 744.843,A -85,B 0,C 180,E1 -14015.638,E2 -14015.638} C_VEL
LIN {X 0,Y 340.738,Z 744.85,A -85,B 0,C 180,E1 -14019.473,E2 -14019.473} C_VEL
LIN {X 0,Y 340.794,Z 744.827,A -85,B 0,C 180,E1 -14021.981,E2 -14021.981} C_VEL
LIN {X 0,Y 340.871,Z 744.835,A -85,B 0,C 180,E1 -14025.705,E2 -14025.705} C_VEL
LIN {X 0,Y 340.873,Z 744.832,A -85,B 0,C 180,E1 -14029.306,E2 -14029.306} C_VEL
LIN {X 0,Y 341.076,Z 744.784,A -85,B 0,C 180,E1 -14032.898,E2 -14032.898} C_VEL
LIN {X 0,Y 341.172,Z 744.8,A -85,B 0,C 180,E1 -14037.639,E2 -14037.639} C_VEL
LIN {X 0,Y 341.297,Z 744.772,A -85,B 0,C 180,E1 -14040,E2 -14040} C_VEL
LIN {X 0,Y 341.17,Z 744.772,A -85,B 0,C 180,E1 -14042.361,E2 -14042.361} C_VEL
LIN {X 0,Y 341.06,Z 744.812,A -85,B 0,C 180,E1 -14047.102,E2 -14047.102} C_VEL
LIN {X 0,Y 340.873,Z 744.822,A -85,B 0,C 180,E1 -14050.694,E2 -14050.694} C_VEL
LIN {X 0,Y 340.864,Z 744.831,A -85,B 0,C 180,E1 -14054.325,E2 -14054.325} C_VEL
LIN {X 0,Y 340.84,Z 744.835,A -85,B 0,C 180,E1 -14058.467,E2 -14058.467} C_VEL
LIN {X 0,Y 340.755,Z 744.832,A -85,B 0,C 180,E1 -14061.857,E2 -14061.857} C_VEL
LIN {X 0,Y 340.773,Z 744.849,A -85,B 0,C 180,E1 -14065.664,E2 -14065.664} C_VEL
LIN {X 0,Y 340.729,Z 744.841,A -85,B 0,C 180,E1 -14068.321,E2 -14068.321} C_VEL
LIN {X 0,Y 340.698,Z 744.851,A -85,B 0,C 180,E1 -14071.044,E2 -14071.044} C_VEL
LIN {X 0,Y 340.719,Z 744.848,A -85,B 0,C 180,E1 -14075.279,E2 -14075.279} C_VEL
LIN {X 0,Y 340.715,Z 744.807,A -85,B 0,C 180,E1 -14078.387,E2 -14078.387} C_VEL
LIN {X 0,Y 340.731,Z 744.835,A -85,B 0,C 180,E1 -14082.051,E2 -14082.051} C_VEL
LIN {X 0,Y 340.659,Z 744.86,A -85,B 0,C 180,E1 -14086.226,E2 -14086.226} C_VEL
LIN {X 0,Y 340.689,Z 744.847,A -85,B 0,C 180,E1 -14089.753,E2 -14089.753} C_VEL
LIN {X 0,Y 340.708,Z 744.849,A -85,B 0,C 180,E1 -14093.259,E2 -14093.259} C_VEL
LIN {X 0,Y 340.695,Z 744.86,A -85,B 0,C 180,E1 -14096.154,E2 -14096.154} C_VEL
LIN {X 0,Y 340.775,Z 744.828,A -85,B 0,C 180,E1 -14100.332,E2 -14100.332} C_VEL
LIN {X 0,Y 340.801,Z 744.916,A -85,B 0,C 180,E1 -14102.467,E2 -14102.467} C_VEL
LIN {X 0,Y 342.468,Z 753.423,A -85,B 0,C 180,E1 -14105.239,E2 -14105.239} C_VEL
LIN {X 0,Y 343.21,Z 758.402,A -85,B 0,C 180,E1 -14106.785,E2 -14106.785} C_VEL
LIN {X 0,Y 342.202,Z 769.043,A -85,B 0,C 180,E1 -14109.879,E2 -14109.879} C_VEL
LIN {X 0,Y 341.724,Z 774.984,A -85,B 0,C 180,E1 -14111.513,E2 -14111.513} C_VEL
LIN {X 0,Y 343.611,Z 786.868,A -85,B 0,C 180,E1 -14111.917,E2 -14111.917} C_VEL
LIN {X 0,Y 346.08,Z 806.281,A -85,B 0,C 180,E1 -14112.463,E2 -14112.463} C_VEL
LIN {X 0,Y 345.447,Z 852.435,A -85,B 0,C 180,E1 -14113.452,E2 -14113.452} C_VEL
LIN {X 0,Y 344.906,Z 863.659,A -85,B 0,C 180,E1 -14113.881,E2 -14113.881} C_VEL
LIN {X 0,Y 344.168,Z 875.393,A -85,B 0,C 180,E1 -14114.606,E2 -14114.606} C_VEL
LIN {X 0,Y 343.468,Z 884.097,A -85,B 0,C 180,E1 -14115.332,E2 -14115.332} C_VEL
LIN {X 0,Y 342.723,Z 892.412,A -85,B 0,C 180,E1 -14116.209,E2 -14116.209} C_VEL
LIN {X 0,Y 341.908,Z 900.282,A -85,B 0,C 180,E1 -14117.234,E2 -14117.234} C_VEL
LIN {X 0,Y 341.185,Z 907.645,A -85,B 0,C 180,E1 -14118.414,E2 -14118.414} C_VEL
LIN {X 0,Y 340.442,Z 915.117,A -85,B 0,C 180,E1 -14119.894,E2 -14119.894} C_VEL
LIN {X 0,Y 339.77,Z 921.941,A -85,B 0,C 180,E1 -14121.675,E2 -14121.675} C_VEL
LIN {X 0,Y 339.36,Z 927.279,A -85,B 0,C 180,E1 -14123.519,E2 -14123.519} C_VEL
LIN {X 0,Y 339.18,Z 930.936,A -85,B 0,C 180,E1 -14125.246,E2 -14125.246} C_VEL
LIN {X 0,Y 339.103,Z 932.688,A -85,B 0,C 180,E1 -14126.435,E2 -14126.435} C_VEL
LIN {X 0,Y 339.003,Z 933.941,A -85,B 0,C 180,E1 -14127.624,E2 -14127.624} C_VEL
LIN {X 0,Y 339.017,Z 934.722,A -85,B 0,C 180,E1 -14128.812,E2 -14128.812} C_VEL
LIN {X 0,Y 339.066,Z 935.019,A -85,B 0,C 180,E1 -14130,E2 -14130} C_VEL
LIN {X 0,Y 339.017,Z 934.719,A -85,B 0,C 180,E1 -14131.188,E2 -14131.188} C_VEL
LIN {X 0,Y 339.003,Z 933.931,A -85,B 0,C 180,E1 -14132.376,E2 -14132.376} C_VEL
LIN {X 0,Y 339.103,Z 932.671,A -85,B 0,C 180,E1 -14133.565,E2 -14133.565} C_VEL
LIN {X 0,Y 339.18,Z 930.912,A -85,B 0,C 180,E1 -14134.754,E2 -14134.754} C_VEL
LIN {X 0,Y 339.364,Z 927.248,A -85,B 0,C 180,E1 -14136.481,E2 -14136.481} C_VEL
LIN {X 0,Y 339.77,Z 921.899,A -85,B 0,C 180,E1 -14138.325,E2 -14138.325} C_VEL
LIN {X 0,Y 340.427,Z 915.055,A -85,B 0,C 180,E1 -14140.107,E2 -14140.107} C_VEL
LIN {X 0,Y 341.186,Z 907.577,A -85,B 0,C 180,E1 -14141.586,E2 -14141.586} C_VEL
LIN {X 0,Y 341.899,Z 900.203,A -85,B 0,C 180,E1 -14142.766,E2 -14142.766} C_VEL
LIN {X 0,Y 342.712,Z 892.311,A -85,B 0,C 180,E1 -14143.792,E2 -14143.792} C_VEL
LIN {X 0,Y 343.492,Z 883.971,A -85,B 0,C 180,E1 -14144.667,E2 -14144.667} C_VEL
LIN {X 0,Y 344.281,Z 873.316,A -85,B 0,C 180,E1 -14145.541,E2 -14145.541} C_VEL
LIN {X 0,Y 344.902,Z 862.544,A -85,B 0,C 180,E1 -14146.157,E2 -14146.157} C_VEL
LIN {X 0,Y 345.461,Z 851.989,A -85,B 0,C 180,E1 -14146.548,E2 -14146.548} C_VEL
LIN {X 0,Y 345.97,Z 804.432,A -85,B 0,C 180,E1 -14147.569,E2 -14147.569} C_VEL
LIN {X 0,Y 342.498,Z 780.094,A -85,B 0,C 180,E1 -14148.276,E2 -14148.276} C_VEL
LIN {X 0,Y 341.698,Z 775.033,A -85,B 0,C 180,E1 -14148.469,E2 -14148.469} C_VEL
LIN {X 0,Y 341.995,Z 771.125,A -85,B 0,C 180,E1 -14149.508,E2 -14149.508} C_VEL
LIN {X 0,Y 343.15,Z 759.428,A -85,B 0,C 180,E1 -14152.901,E2 -14152.901} C_VEL
LIN {X 0,Y 342.734,Z 755.119,A -85,B 0,C 180,E1 -14154.212,E2 -14154.212} C_VEL
LIN {X 0,Y 340.854,Z 745.102,A -85,B 0,C 180,E1 -14157.41,E2 -14157.41} C_VEL
LIN {X 0,Y 340.743,Z 744.856,A -85,B 0,C 180,E1 -14158.32,E2 -14158.32} C_VEL
LIN {X 0,Y 340.704,Z 744.832,A -85,B 0,C 180,E1 -14161.044,E2 -14161.044} C_VEL
LIN {X 0,Y 340.719,Z 744.848,A -85,B 0,C 180,E1 -14165.279,E2 -14165.279} C_VEL
LIN {X 0,Y 340.712,Z 744.855,A -85,B 0,C 180,E1 -14168.387,E2 -14168.387} C_VEL
LIN {X 0,Y 340.699,Z 744.841,A -85,B 0,C 180,E1 -14172.046,E2 -14172.046} C_VEL
LIN {X 0,Y 340.674,Z 744.856,A -85,B 0,C 180,E1 -14176.223,E2 -14176.223} C_VEL
LIN {X 0,Y 340.704,Z 744.827,A -85,B 0,C 180,E1 -14178.693,E2 -14178.693} C_VEL
LIN {X 0,Y 340.738,Z 744.807,A -85,B 0,C 180,E1 -14181.773,E2 -14181.773} C_VEL
LIN {X 0,Y 340.723,Z 744.852,A -85,B 0,C 180,E1 -14185.595,E2 -14185.595} C_VEL
LIN {X 0,Y 340.698,Z 744.851,A -85,B 0,C 180,E1 -14188.956,E2 -14188.956} C_VEL
LIN {X 0,Y 340.804,Z 744.841,A -85,B 0,C 180,E1 -14193.02,E2 -14193.02} C_VEL
LIN {X 0,Y 340.731,Z 744.843,A -85,B 0,C 180,E1 -14196.927,E2 -14196.927} C_VEL
LIN {X 0,Y 340.801,Z 744.84,A -85,B 0,C 180,E1 -14200.734,E2 -14200.734} C_VEL
LIN {X 0,Y 340.788,Z 744.844,A -85,B 0,C 180,E1 -14203.219,E2 -14203.219} C_VEL
LIN {X 0,Y 340.845,Z 744.818,A -85,B 0,C 180,E1 -14206.891,E2 -14206.891} C_VEL
LIN {X 0,Y 340.925,Z 744.825,A -85,B 0,C 180,E1 -14210.508,E2 -14210.508} C_VEL
LIN {X 0,Y 341.061,Z 744.812,A -85,B 0,C 180,E1 -14212.898,E2 -14212.898} C_VEL
LIN {X 0,Y 341.17,Z 744.771,A -85,B 0,C 180,E1 -14217.639,E2 -14217.639} C_VEL
LIN {X 0,Y 341.298,Z 744.771,A -85,B 0,C 180,E1 -14220,E2 -14220} C_VEL
LIN {X 0,Y 341.172,Z 744.799,A -85,B 0,C 180,E1 -14222.361,E2 -14222.361} C_VEL
LIN {X 0,Y 341.076,Z 744.784,A -85,B 0,C 180,E1 -14227.102,E2 -14227.102} C_VEL
LIN {X 0,Y 340.873,Z 744.832,A -85,B 0,C 180,E1 -14230.694,E2 -14230.694} C_VEL
LIN {X 0,Y 340.864,Z 744.835,A -85,B 0,C 180,E1 -14234.325,E2 -14234.325} C_VEL
LIN {X 0,Y 340.787,Z 744.829,A -85,B 0,C 180,E1 -14238.441,E2 -14238.441} C_VEL
LIN {X 0,Y 340.719,Z 744.853,A -85,B 0,C 180,E1 -14241.842,E2 -14241.842} C_VEL
LIN {X 0,Y 340.773,Z 744.828,A -85,B 0,C 180,E1 -14245.664,E2 -14245.664} C_VEL
LIN {X 0,Y 340.73,Z 744.849,A -85,B 0,C 180,E1 -14248.321,E2 -14248.321} C_VEL
LIN {X 0,Y 340.699,Z 744.857,A -85,B 0,C 180,E1 -14251.045,E2 -14251.045} C_VEL
LIN {X 0,Y 340.719,Z 744.851,A -85,B 0,C 180,E1 -14255.279,E2 -14255.279} C_VEL
LIN {X 0,Y 340.711,Z 744.852,A -85,B 0,C 180,E1 -14258.386,E2 -14258.386} C_VEL
LIN {X 0,Y 340.699,Z 744.81,A -85,B 0,C 180,E1 -14262.045,E2 -14262.045} C_VEL
LIN {X 0,Y 340.653,Z 744.861,A -85,B 0,C 180,E1 -14266.227,E2 -14266.227} C_VEL
LIN {X 0,Y 340.689,Z 744.847,A -85,B 0,C 180,E1 -14269.753,E2 -14269.753} C_VEL
LIN {X 0,Y 340.706,Z 744.846,A -85,B 0,C 180,E1 -14273.258,E2 -14273.258} C_VEL
LIN {X 0,Y 340.693,Z 744.858,A -85,B 0,C 180,E1 -14276.153,E2 -14276.153} C_VEL
LIN {X 0,Y 340.725,Z 744.854,A -85,B 0,C 180,E1 -14280.034,E2 -14280.034} C_VEL
LIN {X 0,Y 340.725,Z 744.855,A -85,B 0,C 180,E1 -14283.013,E2 -14283.013} C_VEL
LIN {X 0,Y 340.744,Z 744.852,A -85,B 0,C 180,E1 -14285.637,E2 -14285.637} C_VEL
LIN {X 0,Y 340.805,Z 745.05,A -85,B 0,C 180,E1 -14287.554,E2 -14287.554} C_VEL
LIN {X 0,Y 341.968,Z 752.236,A -85,B 0,C 180,E1 -14290.178,E2 -14290.178} C_VEL
LIN {X 0,Y 341.988,Z 756.421,A -85,B 0,C 180,E1 -14291.568,E2 -14291.568} C_VEL
LIN {X 0,Y 342.365,Z 758.623,A -85,B 0,C 180,E1 -14291.711,E2 -14291.711} C_VEL
LIN {X 0,Y 346.397,Z 779.767,A -85,B 0,C 180,E1 -14292.386,E2 -14292.386} C_VEL
LIN {X 0,Y 345.643,Z 832.253,A -85,B 0,C 180,E1 -14293.499,E2 -14293.499} C_VEL
LIN {X 0,Y 345.394,Z 841.218,A -85,B 0,C 180,E1 -14293.829,E2 -14293.829} C_VEL
LIN {X 0,Y 344.865,Z 850.747,A -85,B 0,C 180,E1 -14294.334,E2 -14294.334} C_VEL
LIN {X 0,Y 344.256,Z 860.746,A -85,B 0,C 180,E1 -14295.064,E2 -14295.064} C_VEL
LIN {X 0,Y 343.323,Z 871.116,A -85,B 0,C 180,E1 -14296.082,E2 -14296.082} C_VEL
LIN {X 0,Y 342.656,Z 879.238,A -85,B 0,C 180,E1 -14297.112,E2 -14297.112} C_VEL
LIN {X 0,Y 341.984,Z 885.94,A -85,B 0,C 180,E1 -14298.141,E2 -14298.141} C_VEL
LIN {X 0,Y 341.294,Z 892.284,A -85,B 0,C 180,E1 -14299.32,E2 -14299.32} C_VEL
LIN {X 0,Y 340.696,Z 897.557,A -85,B 0,C 180,E1 -14300.501,E2 -14300.501} C_VEL
LIN {X 0,Y 340.262,Z 901.957,A -85,B 0,C 180,E1 -14301.687,E2 -14301.687} C_VEL
LIN {X 0,Y 339.916,Z 905.806,A -85,B 0,C 180,E1 -14302.948,E2 -14302.948} C_VEL
LIN {X 0,Y 339.562,Z 909.782,A -85,B 0,C 180,E1 -14304.656,E2 -14304.656} C_VEL
LIN {X 0,Y 339.229,Z 912.69,A -85,B 0,C 180,E1 -14306.437,E2 -14306.437} C_VEL
LIN {X 0,Y 339.123,Z 913.959,A -85,B 0,C 180,E1 -14307.625,E2 -14307.625} C_VEL
LIN {X 0,Y 339.066,Z 914.76,A -85,B 0,C 180,E1 -14308.812,E2 -14308.812} C_VEL
LIN {X 0,Y 339.071,Z 915.064,A -85,B 0,C 180,E1 -14310,E2 -14310} C_VEL
LIN {X 0,Y 339.064,Z 914.787,A -85,B 0,C 180,E1 -14311.188,E2 -14311.188} C_VEL
LIN {X 0,Y 339.112,Z 914.042,A -85,B 0,C 180,E1 -14312.376,E2 -14312.376} C_VEL
LIN {X 0,Y 339.227,Z 912.829,A -85,B 0,C 180,E1 -14313.563,E2 -14313.563} C_VEL
LIN {X 0,Y 339.549,Z 909.979,A -85,B 0,C 180,E1 -14315.344,E2 -14315.344} C_VEL
LIN {X 0,Y 339.906,Z 906.101,A -85,B 0,C 180,E1 -14317.038,E2 -14317.038} C_VEL
LIN {X 0,Y 340.409,Z 900.297,A -85,B 0,C 180,E1 -14318.908,E2 -14318.908} C_VEL
LIN {X 0,Y 341.085,Z 894.185,A -85,B 0,C 180,E1 -14320.387,E2 -14320.387} C_VEL
LIN {X 0,Y 341.739,Z 888.215,A -85,B 0,C 180,E1 -14321.567,E2 -14321.567} C_VEL
LIN {X 0,Y 342.486,Z 880.946,A -85,B 0,C 180,E1 -14322.744,E2 -14322.744} C_VEL
LIN {X 0,Y 343.232,Z 873.176,A -85,B 0,C 180,E1 -14323.77,E2 -14323.77} C_VEL
LIN {X 0,Y 343.855,Z 866.472,A -85,B 0,C 180,E1 -14324.5,E2 -14324.5} C_VEL
LIN {X 0,Y 344.474,Z 858.279,A -85,B 0,C 180,E1 -14325.229,E2 -14325.229} C_VEL
LIN {X 0,Y 344.991,Z 849.971,A -85,B 0,C 180,E1 -14325.811,E2 -14325.811} C_VEL
LIN {X 0,Y 345.381,Z 840.986,A -85,B 0,C 180,E1 -14326.286,E2 -14326.286} C_VEL
LIN {X 0,Y 345.659,Z 831.711,A -85,B 0,C 180,E1 -14326.619,E2 -14326.619} C_VEL
LIN {X 0,Y 346.31,Z 779.011,A -85,B 0,C 180,E1 -14327.738,E2 -14327.738} C_VEL
LIN {X 0,Y 341.985,Z 756.378,A -85,B 0,C 180,E1 -14328.496,E2 -14328.496} C_VEL
LIN {X 0,Y 341.81,Z 750.735,A -85,B 0,C 180,E1 -14330.459,E2 -14330.459} C_VEL
LIN {X 0,Y 340.827,Z 744.948,A -85,B 0,C 180,E1 -14332.609,E2 -14332.609} C_VEL
LIN {X 0,Y 340.722,Z 744.855,A -85,B 0,C 180,E1 -14335.668,E2 -14335.668} C_VEL
LIN {X 0,Y 340.682,Z 744.858,A -85,B 0,C 180,E1 -14338.078,E2 -14338.078} C_VEL
LIN {X 0,Y 340.025,Z 744.942,A -85,B 0,C 180,E1 -14339.064,E2 -14339.064} C_VEL
LIN {X 0,Y 337.191,Z 745.293,A -85,B 0,C 180,E1 -14340.669,E2 -14340.669} C_VEL
LIN {X 0,Y 334.776,Z 745.593,A -85,B 0,C 180,E1 -14341.968,E2 -14341.968} C_VEL
LIN {X 0,Y 333.726,Z 745.722,A -85,B 0,C 180,E1 -14342.973,E2 -14342.973} C_VEL
LIN {X 0,Y 333.633,Z 745.733,A -85,B 0,C 180,E1 -14343.314,E2 -14343.314} C_VEL
LIN {X 0,Y 333.666,Z 745.723,A -85,B 0,C 180,E1 -14346.832,E2 -14346.832} C_VEL
LIN {X 0,Y 333.648,Z 745.729,A -85,B 0,C 180,E1 -14350.767,E2 -14350.767} C_VEL
LIN {X 0,Y 333.594,Z 745.736,A -85,B 0,C 180,E1 -14354.25,E2 -14354.25} C_VEL
LIN {X 0,Y 333.642,Z 745.687,A -85,B 0,C 180,E1 -14357.618,E2 -14357.618} C_VEL
LIN {X 0,Y 333.654,Z 745.729,A -85,B 0,C 180,E1 -14361.202,E2 -14361.202} C_VEL
LIN {X 0,Y 333.677,Z 745.731,A -85,B 0,C 180,E1 -14363.861,E2 -14363.861} C_VEL
LIN {X 0,Y 333.644,Z 745.726,A -85,B 0,C 180,E1 -14367.413,E2 -14367.413} C_VEL
LIN {X 0,Y 333.691,Z 745.731,A -85,B 0,C 180,E1 -14371.026,E2 -14371.026} C_VEL
LIN {X 0,Y 333.736,Z 745.705,A -85,B 0,C 180,E1 -14373.754,E2 -14373.754} C_VEL
LIN {X 0,Y 333.658,Z 745.734,A -85,B 0,C 180,E1 -14377.719,E2 -14377.719} C_VEL
LIN {X 0,Y 333.743,Z 745.707,A -85,B 0,C 180,E1 -14381.586,E2 -14381.586} C_VEL
LIN {X 0,Y 333.809,Z 745.713,A -85,B 0,C 180,E1 -14385.577,E2 -14385.577} C_VEL
LIN {X 0,Y 333.835,Z 745.712,A -85,B 0,C 180,E1 -14389.078,E2 -14389.078} C_VEL
LIN {X 0,Y 334.026,Z 745.661,A -85,B 0,C 180,E1 -14392.747,E2 -14392.747} C_VEL
LIN {X 0,Y 333.813,Z 745.707,A -85,B 0,C 180,E1 -14395.169,E2 -14395.169} C_VEL
LIN {X 0,Y 334.133,Z 745.677,A -85,B 0,C 180,E1 -14397.589,E2 -14397.589} C_VEL
LIN {X 0,Y 334.247,Z 745.65,A -85,B 0,C 180,E1 -14400,E2 -14400} C_VEL
LIN {X 0,Y 334.107,Z 745.651,A -85,B 0,C 180,E1 -14402.411,E2 -14402.411} C_VEL
LIN {X 0,Y 334.016,Z 745.69,A -85,B 0,C 180,E1 -14406.039,E2 -14406.039} C_VEL
LIN {X 0,Y 333.861,Z 745.702,A -85,B 0,C 180,E1 -14409.695,E2 -14409.695} C_VEL
LIN {X 0,Y 333.798,Z 745.697,A -85,B 0,C 180,E1 -14413.391,E2 -14413.391} C_VEL
LIN {X 0,Y 333.748,Z 745.722,A -85,B 0,C 180,E1 -14417.146,E2 -14417.146} C_VEL
LIN {X 0,Y 333.749,Z 745.712,A -85,B 0,C 180,E1 -14419.689,E2 -14419.689} C_VEL
LIN {X 0,Y 333.682,Z 745.724,A -85,B 0,C 180,E1 -14423.589,E2 -14423.589} C_VEL
LIN {X 0,Y 333.736,Z 745.725,A -85,B 0,C 180,E1 -14426.246,E2 -14426.246} C_VEL
LIN {X 0,Y 333.691,Z 745.713,A -85,B 0,C 180,E1 -14428.974,E2 -14428.974} C_VEL
LIN {X 0,Y 333.646,Z 745.737,A -85,B 0,C 180,E1 -14432.587,E2 -14432.587} C_VEL
LIN {X 0,Y 333.678,Z 745.715,A -85,B 0,C 180,E1 -14436.139,E2 -14436.139} C_VEL
LIN {X 0,Y 333.671,Z 745.678,A -85,B 0,C 180,E1 -14439.189,E2 -14439.189} C_VEL
LIN {X 0,Y 333.666,Z 745.72,A -85,B 0,C 180,E1 -14442.506,E2 -14442.506} C_VEL
LIN {X 0,Y 333.609,Z 745.741,A -85,B 0,C 180,E1 -14445.957,E2 -14445.957} C_VEL
LIN {X 0,Y 333.647,Z 745.719,A -85,B 0,C 180,E1 -14449.315,E2 -14449.315} C_VEL
LIN {X 0,Y 333.667,Z 745.726,A -85,B 0,C 180,E1 -14453.167,E2 -14453.167} C_VEL
LIN {X 0,Y 333.639,Z 745.736,A -85,B 0,C 180,E1 -14456.792,E2 -14456.792} C_VEL
LIN {X 0,Y 333.703,Z 745.703,A -85,B 0,C 180,E1 -14459.71,E2 -14459.71} C_VEL
LIN {X 0,Y 333.756,Z 745.893,A -85,B 0,C 180,E1 -14462.231,E2 -14462.231} C_VEL
LIN {X 0,Y 335.722,Z 756.061,A -85,B 0,C 180,E1 -14465.578,E2 -14465.578} C_VEL
LIN {X 0,Y 336.21,Z 760.231,A -85,B 0,C 180,E1 -14466.891,E2 -14466.891} C_VEL
LIN {X 0,Y 334.818,Z 774.236,A -85,B 0,C 180,E1 -14471.012,E2 -14471.012} C_VEL
LIN {X 0,Y 334.792,Z 774.943,A -85,B 0,C 180,E1 -14471.13,E2 -14471.13} C_VEL
LIN {X 0,Y 337.974,Z 795.669,A -85,B 0,C 180,E1 -14471.801,E2 -14471.801} C_VEL
LIN {X 0,Y 339.311,Z 807.286,A -85,B 0,C 180,E1 -14472.127,E2 -14472.127} C_VEL
LIN {X 0,Y 338.658,Z 852.241,A -85,B 0,C 180,E1 -14473.11,E2 -14473.11} C_VEL
LIN {X 0,Y 338.108,Z 863.46,A -85,B 0,C 180,E1 -14473.548,E2 -14473.548} C_VEL
LIN {X 0,Y 337.329,Z 875.189,A -85,B 0,C 180,E1 -14474.285,E2 -14474.285} C_VEL
LIN {X 0,Y 336.607,Z 883.892,A -85,B 0,C 180,E1 -14475.026,E2 -14475.026} C_VEL
LIN {X 0,Y 335.837,Z 892.207,A -85,B 0,C 180,E1 -14475.92,E2 -14475.92} C_VEL
LIN {X 0,Y 334.992,Z 900.076,A -85,B 0,C 180,E1 -14476.966,E2 -14476.966} C_VEL
LIN {X 0,Y 334.224,Z 907.439,A -85,B 0,C 180,E1 -14478.169,E2 -14478.169} C_VEL
LIN {X 0,Y 333.415,Z 914.909,A -85,B 0,C 180,E1 -14479.679,E2 -14479.679} C_VEL
LIN {X 0,Y 332.73,Z 921.733,A -85,B 0,C 180,E1 -14481.497,E2 -14481.497} C_VEL
LIN {X 0,Y 332.315,Z 926.918,A -85,B 0,C 180,E1 -14483.32,E2 -14483.32} C_VEL
LIN {X 0,Y 332.083,Z 930.728,A -85,B 0,C 180,E1 -14485.144,E2 -14485.144} C_VEL
LIN {X 0,Y 332.031,Z 932.48,A -85,B 0,C 180,E1 -14486.359,E2 -14486.359} C_VEL
LIN {X 0,Y 331.922,Z 933.733,A -85,B 0,C 180,E1 -14487.573,E2 -14487.573} C_VEL
LIN {X 0,Y 331.922,Z 934.514,A -85,B 0,C 180,E1 -14488.787,E2 -14488.787} C_VEL
LIN {X 0,Y 331.968,Z 934.81,A -85,B 0,C 180,E1 -14490,E2 -14490} C_VEL
LIN {X 0,Y 331.922,Z 934.51,A -85,B 0,C 180,E1 -14491.213,E2 -14491.213} C_VEL
LIN {X 0,Y 331.922,Z 933.722,A -85,B 0,C 180,E1 -14492.427,E2 -14492.427} C_VEL
LIN {X 0,Y 332.031,Z 932.462,A -85,B 0,C 180,E1 -14493.641,E2 -14493.641} C_VEL
LIN {X 0,Y 332.083,Z 930.702,A -85,B 0,C 180,E1 -14494.856,E2 -14494.856} C_VEL
LIN {X 0,Y 332.316,Z 926.885,A -85,B 0,C 180,E1 -14496.68,E2 -14496.68} C_VEL
LIN {X 0,Y 332.73,Z 921.688,A -85,B 0,C 180,E1 -14498.503,E2 -14498.503} C_VEL
LIN {X 0,Y 333.4,Z 914.843,A -85,B 0,C 180,E1 -14500.322,E2 -14500.322} C_VEL
LIN {X 0,Y 334.224,Z 907.365,A -85,B 0,C 180,E1 -14501.831,E2 -14501.831} C_VEL
LIN {X 0,Y 334.985,Z 899.992,A -85,B 0,C 180,E1 -14503.034,E2 -14503.034} C_VEL
LIN {X 0,Y 335.833,Z 892.099,A -85,B 0,C 180,E1 -14504.08,E2 -14504.08} C_VEL
LIN {X 0,Y 336.643,Z 883.758,A -85,B 0,C 180,E1 -14504.972,E2 -14504.972} C_VEL
LIN {X 0,Y 337.443,Z 873.101,A -85,B 0,C 180,E1 -14505.864,E2 -14505.864} C_VEL
LIN {X 0,Y 338.094,Z 862.326,A -85,B 0,C 180,E1 -14506.492,E2 -14506.492} C_VEL
LIN {X 0,Y 338.607,Z 853.063,A -85,B 0,C 180,E1 -14506.854,E2 -14506.854} C_VEL
LIN {X 0,Y 338.946,Z 826.753,A -85,B 0,C 180,E1 -14507.455,E2 -14507.455} C_VEL
LIN {X 0,Y 339.246,Z 805.474,A -85,B 0,C 180,E1 -14507.902,E2 -14507.902} C_VEL
LIN {X 0,Y 335.489,Z 779.345,A -85,B 0,C 180,E1 -14508.683,E2 -14508.683} C_VEL
LIN {X 0,Y 334.783,Z 774.794,A -85,B 0,C 180,E1 -14508.867,E2 -14508.867} C_VEL
LIN {X 0,Y 335.308,Z 768.799,A -85,B 0,C 180,E1 -14510.553,E2 -14510.553} C_VEL
LIN {X 0,Y 336.209,Z 759.229,A -85,B 0,C 180,E1 -14513.401,E2 -14513.401} C_VEL
LIN {X 0,Y 334.703,Z 750.609,A -85,B 0,C 180,E1 -14516.165,E2 -14516.165} C_VEL
LIN {X 0,Y 333.739,Z 745.751,A -85,B 0,C 180,E1 -14517.846,E2 -14517.846} C_VEL
LIN {X 0,Y 333.697,Z 745.704,A -85,B 0,C 180,E1 -14520.362,E2 -14520.362} C_VEL
LIN {X 0,Y 333.674,Z 745.732,A -85,B 0,C 180,E1 -14524.659,E2 -14524.659} C_VEL
LIN {X 0,Y 333.655,Z 745.737,A -85,B 0,C 180,E1 -14527.651,E2 -14527.651} C_VEL
LIN {X 0,Y 333.647,Z 745.718,A -85,B 0,C 180,E1 -14530.767,E2 -14530.767} C_VEL
LIN {X 0,Y 333.609,Z 745.74,A -85,B 0,C 180,E1 -14534.253,E2 -14534.253} C_VEL
LIN {X 0,Y 333.674,Z 745.716,A -85,B 0,C 180,E1 -14537.624,E2 -14537.624} C_VEL
LIN {X 0,Y 333.675,Z 745.679,A -85,B 0,C 180,E1 -14541.197,E2 -14541.197} C_VEL
LIN {X 0,Y 333.686,Z 745.726,A -85,B 0,C 180,E1 -14545.226,E2 -14545.226} C_VEL
LIN {X 0,Y 333.632,Z 745.734,A -85,B 0,C 180,E1 -14548.222,E2 -14548.222} C_VEL
LIN {X 0,Y 333.691,Z 745.714,A -85,B 0,C 180,E1 -14551.026,E2 -14551.026} C_VEL
LIN {X 0,Y 333.736,Z 745.725,A -85,B 0,C 180,E1 -14553.754,E2 -14553.754} C_VEL
LIN {X 0,Y 333.72,Z 745.709,A -85,B 0,C 180,E1 -14557.914,E2 -14557.914} C_VEL
LIN {X 0,Y 333.796,Z 745.713,A -85,B 0,C 180,E1 -14561.59,E2 -14561.59} C_VEL
LIN {X 0,Y 333.809,Z 745.709,A -85,B 0,C 180,E1 -14565.577,E2 -14565.577} C_VEL
LIN {X 0,Y 333.835,Z 745.699,A -85,B 0,C 180,E1 -14569.078,E2 -14569.078} C_VEL
LIN {X 0,Y 334.008,Z 745.691,A -85,B 0,C 180,E1 -14572.747,E2 -14572.747} C_VEL
LIN {X 0,Y 333.811,Z 745.705,A -85,B 0,C 180,E1 -14575.169,E2 -14575.169} C_VEL
LIN {X 0,Y 334.107,Z 745.65,A -85,B 0,C 180,E1 -14577.589,E2 -14577.589} C_VEL
LIN {X 0,Y 334.249,Z 745.649,A -85,B 0,C 180,E1 -14580,E2 -14580} C_VEL
LIN {X 0,Y 334.133,Z 745.676,A -85,B 0,C 180,E1 -14582.411,E2 -14582.411} C_VEL
LIN {X 0,Y 334.026,Z 745.661,A -85,B 0,C 180,E1 -14587.253,E2 -14587.253} C_VEL
LIN {X 0,Y 333.835,Z 745.711,A -85,B 0,C 180,E1 -14590.922,E2 -14590.922} C_VEL
LIN {X 0,Y 333.809,Z 745.711,A -85,B 0,C 180,E1 -14594.634,E2 -14594.634} C_VEL
LIN {X 0,Y 333.755,Z 745.707,A -85,B 0,C 180,E1 -14598.633,E2 -14598.633} C_VEL
LIN {X 0,Y 333.658,Z 745.734,A -85,B 0,C 180,E1 -14602.281,E2 -14602.281} C_VEL
LIN {X 0,Y 333.736,Z 745.705,A -85,B 0,C 180,E1 -14606.246,E2 -14606.246} C_VEL
LIN {X 0,Y 333.691,Z 745.73,A -85,B 0,C 180,E1 -14608.974,E2 -14608.974} C_VEL
LIN {X 0,Y 333.644,Z 745.727,A -85,B 0,C 180,E1 -14612.587,E2 -14612.587} C_VEL
LIN {X 0,Y 333.677,Z 745.731,A -85,B 0,C 180,E1 -14616.139,E2 -14616.139} C_VEL
LIN {X 0,Y 333.647,Z 745.725,A -85,B 0,C 180,E1 -14619.192,E2 -14619.192} C_VEL
LIN {X 0,Y 333.633,Z 745.687,A -85,B 0,C 180,E1 -14622.5,E2 -14622.5} C_VEL
LIN {X 0,Y 333.598,Z 745.737,A -85,B 0,C 180,E1 -14625.955,E2 -14625.955} C_VEL
LIN {X 0,Y 333.648,Z 745.73,A -85,B 0,C 180,E1 -14629.315,E2 -14629.315} C_VEL
LIN {X 0,Y 333.666,Z 745.722,A -85,B 0,C 180,E1 -14633.168,E2 -14633.168} C_VEL
LIN {X 0,Y 333.675,Z 745.738,A -85,B 0,C 180,E1 -14635.341,E2 -14635.341} C_VEL
LIN {X 0,Y 333.63,Z 745.722,A -85,B 0,C 180,E1 -14638.222,E2 -14638.222} C_VEL
LIN {X 0,Y 333.656,Z 745.736,A -85,B 0,C 180,E1 -14641.023,E2 -14641.023} C_VEL
LIN {X 0,Y 333.7,Z 745.731,A -85,B 0,C 180,E1 -14645.089,E2 -14645.089} C_VEL
LIN {X 0,Y 333.75,Z 745.96,A -85,B 0,C 180,E1 -14647.318,E2 -14647.318} C_VEL
LIN {X 0,Y 334.896,Z 752.436,A -85,B 0,C 180,E1 -14649.741,E2 -14649.741} C_VEL
LIN {X 0,Y 335.02,Z 756.55,A -85,B 0,C 180,E1 -14651.155,E2 -14651.155} C_VEL
LIN {X 0,Y 335.341,Z 758.282,A -85,B 0,C 180,E1 -14651.299,E2 -14651.299} C_VEL
LIN {X 0,Y 339.647,Z 780.453,A -85,B 0,C 180,E1 -14652.034,E2 -14652.034} C_VEL
LIN {X 0,Y 338.85,Z 832.48,A -85,B 0,C 180,E1 -14653.159,E2 -14653.159} C_VEL
LIN {X 0,Y 338.605,Z 841.438,A -85,B 0,C 180,E1 -14653.495,E2 -14653.495} C_VEL
LIN {X 0,Y 338.06,Z 850.964,A -85,B 0,C 180,E1 -14654.011,E2 -14654.011} C_VEL
LIN {X 0,Y 337.411,Z 860.961,A -85,B 0,C 180,E1 -14654.754,E2 -14654.754} C_VEL
LIN {X 0,Y 336.434,Z 871.33,A -85,B 0,C 180,E1 -14655.791,E2 -14655.791} C_VEL
LIN {X 0,Y 335.757,Z 879.45,A -85,B 0,C 180,E1 -14656.842,E2 -14656.842} C_VEL
LIN {X 0,Y 335.045,Z 886.151,A -85,B 0,C 180,E1 -14657.892,E2 -14657.892} C_VEL
LIN {X 0,Y 334.311,Z 892.496,A -85,B 0,C 180,E1 -14659.094,E2 -14659.094} C_VEL
LIN {X 0,Y 333.568,Z 898.936,A -85,B 0,C 180,E1 -14660.602,E2 -14660.602} C_VEL
LIN {X 0,Y 333.077,Z 904.07,A -85,B 0,C 180,E1 -14662.117,E2 -14662.117} C_VEL
LIN {X 0,Y 332.611,Z 908.82,A -85,B 0,C 180,E1 -14663.935,E2 -14663.935} C_VEL
LIN {X 0,Y 332.397,Z 911.136,A -85,B 0,C 180,E1 -14665.148,E2 -14665.148} C_VEL
LIN {X 0,Y 332.16,Z 912.899,A -85,B 0,C 180,E1 -14666.361,E2 -14666.361} C_VEL
LIN {X 0,Y 332.037,Z 914.168,A -85,B 0,C 180,E1 -14667.574,E2 -14667.574} C_VEL
LIN {X 0,Y 331.971,Z 914.969,A -85,B 0,C 180,E1 -14668.787,E2 -14668.787} C_VEL
LIN {X 0,Y 331.974,Z 915.273,A -85,B 0,C 180,E1 -14670,E2 -14670} C_VEL
LIN {X 0,Y 331.97,Z 914.996,A -85,B 0,C 180,E1 -14671.213,E2 -14671.213} C_VEL
LIN {X 0,Y 332.026,Z 914.25,A -85,B 0,C 180,E1 -14672.426,E2 -14672.426} C_VEL
LIN {X 0,Y 332.158,Z 913.037,A -85,B 0,C 180,E1 -14673.639,E2 -14673.639} C_VEL
LIN {X 0,Y 332.484,Z 910.187,A -85,B 0,C 180,E1 -14675.458,E2 -14675.458} C_VEL
LIN {X 0,Y 332.82,Z 906.699,A -85,B 0,C 180,E1 -14677.031,E2 -14677.031} C_VEL
LIN {X 0,Y 333.174,Z 902.495,A -85,B 0,C 180,E1 -14678.491,E2 -14678.491} C_VEL
LIN {X 0,Y 333.78,Z 897.003,A -85,B 0,C 180,E1 -14680.004,E2 -14680.004} C_VEL
LIN {X 0,Y 334.638,Z 890.098,A -85,B 0,C 180,E1 -14681.509,E2 -14681.509} C_VEL
LIN {X 0,Y 335.512,Z 882.168,A -85,B 0,C 180,E1 -14682.86,E2 -14682.86} C_VEL
LIN {X 0,Y 336.263,Z 874.605,A -85,B 0,C 180,E1 -14683.907,E2 -14683.907} C_VEL
LIN {X 0,Y 336.878,Z 868.172,A -85,B 0,C 180,E1 -14684.652,E2 -14684.652} C_VEL
LIN {X 0,Y 337.5,Z 860.351,A -85,B 0,C 180,E1 -14685.397,E2 -14685.397} C_VEL
LIN {X 0,Y 338.122,Z 851.379,A -85,B 0,C 180,E1 -14686.064,E2 -14686.064} C_VEL
LIN {X 0,Y 338.563,Z 842.013,A -85,B 0,C 180,E1 -14686.584,E2 -14686.584} C_VEL
LIN {X 0,Y 338.833,Z 832.91,A -85,B 0,C 180,E1 -14686.934,E2 -14686.934} C_VEL
LIN {X 0,Y 339.575,Z 779.909,A -85,B 0,C 180,E1 -14688.086,E2 -14688.086} C_VEL
LIN {X 0,Y 335.014,Z 756.678,A -85,B 0,C 180,E1 -14688.861,E2 -14688.861} C_VEL
LIN {X 0,Y 334.694,Z 750.933,A -85,B 0,C 180,E1 -14690.914,E2 -14690.914} C_VEL
LIN {X 0,Y 333.768,Z 745.801,A -85,B 0,C 180,E1 -14692.926,E2 -14692.926} C_VEL
LIN {X 0,Y 333.659,Z 745.736,A -85,B 0,C 180,E1 -14696.253,E2 -14696.253} C_VEL
LIN {X 0,Y 333.663,Z 745.73,A -85,B 0,C 180,E1 -14700.278,E2 -14700.278} C_VEL
LIN {X 0,Y 333.633,Z 745.733,A -85,B 0,C 180,E1 -14703.314,E2 -14703.314} C_VEL
LIN {X 0,Y 332.949,Z 745.827,A -85,B 0,C 180,E1 -14704.321,E2 -14704.321} C_VEL
LIN {X 0,Y 330.102,Z 746.179,A -85,B 0,C 180,E1 -14705.96,E2 -14705.96} C_VEL
LIN {X 0,Y 327.704,Z 746.462,A -85,B 0,C 180,E1 -14707.288,E2 -14707.288} C_VEL
LIN {X 0,Y 326.679,Z 746.579,A -85,B 0,C 180,E1 -14708.316,E2 -14708.316} C_VEL
LIN {X 0,Y 326.598,Z 746.589,A -85,B 0,C 180,E1 -14708.664,E2 -14708.664} C_VEL
LIN {X 0,Y 326.577,Z 746.616,A -85,B 0,C 180,E1 -14711.846,E2 -14711.846} C_VEL
LIN {X 0,Y 326.528,Z 746.605,A -85,B 0,C 180,E1 -14715.257,E2 -14715.257} C_VEL
LIN {X 0,Y 326.578,Z 746.576,A -85,B 0,C 180,E1 -14718.869,E2 -14718.869} C_VEL
LIN {X 0,Y 326.629,Z 746.612,A -85,B 0,C 180,E1 -14722.761,E2 -14722.761} C_VEL
LIN {X 0,Y 326.608,Z 746.602,A -85,B 0,C 180,E1 -14725.981,E2 -14725.981} C_VEL
LIN {X 0,Y 326.649,Z 746.607,A -85,B 0,C 180,E1 -14730.34,E2 -14730.34} C_VEL
LIN {X 0,Y 326.691,Z 746.582,A -85,B 0,C 180,E1 -14734.516,E2 -14734.516} C_VEL
LIN {X 0,Y 326.622,Z 746.611,A -85,B 0,C 180,E1 -14738.543,E2 -14738.543} C_VEL
LIN {X 0,Y 326.708,Z 746.587,A -85,B 0,C 180,E1 -14741.175,E2 -14741.175} C_VEL
LIN {X 0,Y 326.764,Z 746.588,A -85,B 0,C 180,E1 -14745.433,E2 -14745.433} C_VEL
LIN {X 0,Y 326.772,Z 746.592,A -85,B 0,C 180,E1 -14748.839,E2 -14748.839} C_VEL
LIN {X 0,Y 326.981,Z 746.537,A -85,B 0,C 180,E1 -14752.59,E2 -14752.59} C_VEL
LIN {X 0,Y 326.78,Z 746.582,A -85,B 0,C 180,E1 -14755.065,E2 -14755.065} C_VEL
LIN {X 0,Y 327.07,Z 746.557,A -85,B 0,C 180,E1 -14757.537,E2 -14757.537} C_VEL
LIN {X 0,Y 327.199,Z 746.527,A -85,B 0,C 180,E1 -14760,E2 -14760} C_VEL
LIN {X 0,Y 327.047,Z 746.53,A -85,B 0,C 180,E1 -14762.463,E2 -14762.463} C_VEL
LIN {X 0,Y 326.99,Z 746.565,A -85,B 0,C 180,E1 -14766.169,E2 -14766.169} C_VEL
LIN {X 0,Y 326.813,Z 746.577,A -85,B 0,C 180,E1 -14769.906,E2 -14769.906} C_VEL
LIN {X 0,Y 326.76,Z 746.576,A -85,B 0,C 180,E1 -14773.685,E2 -14773.685} C_VEL
LIN {X 0,Y 326.702,Z 746.602,A -85,B 0,C 180,E1 -14777.528,E2 -14777.528} C_VEL
LIN {X 0,Y 326.674,Z 746.587,A -85,B 0,C 180,E1 -14780.134,E2 -14780.134} C_VEL
LIN {X 0,Y 326.657,Z 746.605,A -85,B 0,C 180,E1 -14784.128,E2 -14784.128} C_VEL
LIN {X 0,Y 326.684,Z 746.599,A -85,B 0,C 180,E1 -14786.858,E2 -14786.858} C_VEL
LIN {X 0,Y 326.634,Z 746.601,A -85,B 0,C 180,E1 -14790.61,E2 -14790.61} C_VEL
LIN {X 0,Y 326.608,Z 746.614,A -85,B 0,C 180,E1 -14794.019,E2 -14794.019} C_VEL
LIN {X 0,Y 326.631,Z 746.58,A -85,B 0,C 180,E1 -14797.239,E2 -14797.239} C_VEL
LIN {X 0,Y 326.604,Z 746.562,A -85,B 0,C 180,E1 -14800.207,E2 -14800.207} C_VEL
LIN {X 0,Y 326.585,Z 746.611,A -85,B 0,C 180,E1 -14803.522,E2 -14803.522} C_VEL
LIN {X 0,Y 326.579,Z 746.604,A -85,B 0,C 180,E1 -14807.027,E2 -14807.027} C_VEL
LIN {X 0,Y 326.612,Z 746.61,A -85,B 0,C 180,E1 -14810.772,E2 -14810.772} C_VEL
LIN {X 0,Y 326.613,Z 746.602,A -85,B 0,C 180,E1 -14814.48,E2 -14814.48} C_VEL
LIN {X 0,Y 326.61,Z 746.605,A -85,B 0,C 180,E1 -14817.456,E2 -14817.456} C_VEL
LIN {X 0,Y 326.661,Z 746.585,A -85,B 0,C 180,E1 -14820.341,E2 -14820.341} C_VEL
LIN {X 0,Y 326.719,Z 746.828,A -85,B 0,C 180,E1 -14821.951,E2 -14821.951} C_VEL
LIN {X 0,Y 328.696,Z 756.933,A -85,B 0,C 180,E1 -14825.359,E2 -14825.359} C_VEL
LIN {X 0,Y 329.257,Z 760.795,A -85,B 0,C 180,E1 -14826.611,E2 -14826.611} C_VEL
LIN {X 0,Y 327.911,Z 773.918,A -85,B 0,C 180,E1 -14830.568,E2 -14830.568} C_VEL
LIN {X 0,Y 327.905,Z 774.742,A -85,B 0,C 180,E1 -14830.718,E2 -14830.718} C_VEL
LIN {X 0,Y 331.309,Z 797.071,A -85,B 0,C 180,E1 -14831.457,E2 -14831.457} C_VEL
LIN {X 0,Y 332.562,Z 808.299,A -85,B 0,C 180,E1 -14831.778,E2 -14831.778} C_VEL
LIN {X 0,Y 331.873,Z 852.047,A -85,B 0,C 180,E1 -14832.754,E2 -14832.754} C_VEL
LIN {X 0,Y 331.317,Z 863.261,A -85,B 0,C 180,E1 -14833.201,E2 -14833.201} C_VEL
LIN {X 0,Y 330.486,Z 874.985,A -85,B 0,C 180,E1 -14833.951,E2 -14833.951} C_VEL
LIN {X 0,Y 329.763,Z 883.688,A -85,B 0,C 180,E1 -14834.708,E2 -14834.708} C_VEL
LIN {X 0,Y 328.952,Z 892.001,A -85,B 0,C 180,E1 -14835.619,E2 -14835.619} C_VEL
LIN {X 0,Y 328.082,Z 899.87,A -85,B 0,C 180,E1 -14836.686,E2 -14836.686} C_VEL
LIN {X 0,Y 327.269,Z 907.232,A -85,B 0,C 180,E1 -14837.914,E2 -14837.914} C_VEL
LIN {X 0,Y 326.404,Z 914.701,A -85,B 0,C 180,E1 -14839.454,E2 -14839.454} C_VEL
LIN {X 0,Y 325.693,Z 921.525,A -85,B 0,C 180,E1 -14841.312,E2 -14841.312} C_VEL
LIN {X 0,Y 325.264,Z 926.711,A -85,B 0,C 180,E1 -14843.175,E2 -14843.175} C_VEL
LIN {X 0,Y 324.99,Z 930.519,A -85,B 0,C 180,E1 -14845.038,E2 -14845.038} C_VEL
LIN {X 0,Y 324.939,Z 932.272,A -85,B 0,C 180,E1 -14846.28,E2 -14846.28} C_VEL
LIN {X 0,Y 324.843,Z 933.525,A -85,B 0,C 180,E1 -14847.52,E2 -14847.52} C_VEL
LIN {X 0,Y 324.831,Z 934.305,A -85,B 0,C 180,E1 -14848.76,E2 -14848.76} C_VEL
LIN {X 0,Y 324.873,Z 934.601,A -85,B 0,C 180,E1 -14850,E2 -14850} C_VEL
LIN {X 0,Y 324.831,Z 934.301,A -85,B 0,C 180,E1 -14851.24,E2 -14851.24} C_VEL
LIN {X 0,Y 324.843,Z 933.513,A -85,B 0,C 180,E1 -14852.48,E2 -14852.48} C_VEL
LIN {X 0,Y 324.939,Z 932.252,A -85,B 0,C 180,E1 -14853.72,E2 -14853.72} C_VEL
LIN {X 0,Y 325,Z 929.524,A -85,B 0,C 180,E1 -14855.481,E2 -14855.481} C_VEL
LIN {X 0,Y 325.264,Z 926.675,A -85,B 0,C 180,E1 -14856.825,E2 -14856.825} C_VEL
LIN {X 0,Y 325.693,Z 921.477,A -85,B 0,C 180,E1 -14858.688,E2 -14858.688} C_VEL
LIN {X 0,Y 326.394,Z 914.631,A -85,B 0,C 180,E1 -14860.546,E2 -14860.546} C_VEL
LIN {X 0,Y 327.269,Z 907.154,A -85,B 0,C 180,E1 -14862.086,E2 -14862.086} C_VEL
LIN {X 0,Y 328.057,Z 899.779,A -85,B 0,C 180,E1 -14863.315,E2 -14863.315} C_VEL
LIN {X 0,Y 328.953,Z 891.886,A -85,B 0,C 180,E1 -14864.381,E2 -14864.381} C_VEL
LIN {X 0,Y 329.802,Z 883.546,A -85,B 0,C 180,E1 -14865.29,E2 -14865.29} C_VEL
LIN {X 0,Y 330.628,Z 872.886,A -85,B 0,C 180,E1 -14866.2,E2 -14866.2} C_VEL
LIN {X 0,Y 331.309,Z 862.108,A -85,B 0,C 180,E1 -14866.839,E2 -14866.839} C_VEL
LIN {X 0,Y 331.828,Z 852.84,A -85,B 0,C 180,E1 -14867.209,E2 -14867.209} C_VEL
LIN {X 0,Y 332.193,Z 827.795,A -85,B 0,C 180,E1 -14867.793,E2 -14867.793} C_VEL
LIN {X 0,Y 332.387,Z 805.36,A -85,B 0,C 180,E1 -14868.281,E2 -14868.281} C_VEL
LIN {X 0,Y 328.663,Z 779.638,A -85,B 0,C 180,E1 -14869.074,E2 -14869.074} C_VEL
LIN {X 0,Y 327.887,Z 774.514,A -85,B 0,C 180,E1 -14869.287,E2 -14869.287} C_VEL
LIN {X 0,Y 329.165,Z 762.031,A -85,B 0,C 180,E1 -14872.996,E2 -14872.996} C_VEL
LIN {X 0,Y 329.022,Z 759.024,A -85,B 0,C 180,E1 -14873.944,E2 -14873.944} C_VEL
LIN {X 0,Y 327.469,Z 750.416,A -85,B 0,C 180,E1 -14876.788,E2 -14876.788} C_VEL
LIN {X 0,Y 326.679,Z 746.628,A -85,B 0,C 180,E1 -14878.151,E2 -14878.151} C_VEL
LIN {X 0,Y 326.594,Z 746.589,A -85,B 0,C 180,E1 -14881.095,E2 -14881.095} C_VEL
LIN {X 0,Y 326.608,Z 746.615,A -85,B 0,C 180,E1 -14884.019,E2 -14884.019} C_VEL
LIN {X 0,Y 326.63,Z 746.607,A -85,B 0,C 180,E1 -14887.239,E2 -14887.239} C_VEL
LIN {X 0,Y 326.578,Z 746.596,A -85,B 0,C 180,E1 -14891.131,E2 -14891.131} C_VEL
LIN {X 0,Y 326.543,Z 746.62,A -85,B 0,C 180,E1 -14894.746,E2 -14894.746} C_VEL
LIN {X 0,Y 326.598,Z 746.591,A -85,B 0,C 180,E1 -14898.158,E2 -14898.158} C_VEL
LIN {X 0,Y 326.642,Z 746.555,A -85,B 0,C 180,E1 -14901.394,E2 -14901.394} C_VEL
LIN {X 0,Y 326.621,Z 746.605,A -85,B 0,C 180,E1 -14904.851,E2 -14904.851} C_VEL
LIN {X 0,Y 326.61,Z 746.614,A -85,B 0,C 180,E1 -14907.456,E2 -14907.456} C_VEL
LIN {X 0,Y 326.648,Z 746.591,A -85,B 0,C 180,E1 -14910.34,E2 -14910.34} C_VEL
LIN {X 0,Y 326.691,Z 746.602,A -85,B 0,C 180,E1 -14914.516,E2 -14914.516} C_VEL
LIN {X 0,Y 326.653,Z 746.586,A -85,B 0,C 180,E1 -14918.546,E2 -14918.546} C_VEL
LIN {X 0,Y 326.745,Z 746.59,A -85,B 0,C 180,E1 -14921.178,E2 -14921.178} C_VEL
LIN {X 0,Y 326.764,Z 746.586,A -85,B 0,C 180,E1 -14925.433,E2 -14925.433} C_VEL
LIN {X 0,Y 326.771,Z 746.575,A -85,B 0,C 180,E1 -14928.839,E2 -14928.839} C_VEL
LIN {X 0,Y 326.96,Z 746.571,A -85,B 0,C 180,E1 -14932.59,E2 -14932.59} C_VEL
LIN {X 0,Y 326.778,Z 746.582,A -85,B 0,C 180,E1 -14935.065,E2 -14935.065} C_VEL
LIN {X 0,Y 327.048,Z 746.529,A -85,B 0,C 180,E1 -14937.537,E2 -14937.537} C_VEL
LIN {X 0,Y 327.201,Z 746.527,A -85,B 0,C 180,E1 -14940,E2 -14940} C_VEL
LIN {X 0,Y 327.07,Z 746.557,A -85,B 0,C 180,E1 -14942.463,E2 -14942.463} C_VEL
LIN {X 0,Y 326.974,Z 746.544,A -85,B 0,C 180,E1 -14946.6,E2 -14946.6} C_VEL
LIN {X 0,Y 326.815,Z 746.576,A -85,B 0,C 180,E1 -14949.906,E2 -14949.906} C_VEL
LIN {X 0,Y 326.761,Z 746.591,A -85,B 0,C 180,E1 -14953.685,E2 -14953.685} C_VEL
LIN {X 0,Y 326.665,Z 746.584,A -85,B 0,C 180,E1 -14957.53,E2 -14957.53} C_VEL
LIN {X 0,Y 326.651,Z 746.602,A -85,B 0,C 180,E1 -14960.136,E2 -14960.136} C_VEL
LIN {X 0,Y 326.65,Z 746.6,A -85,B 0,C 180,E1 -14964.129,E2 -14964.129} C_VEL
LIN {X 0,Y 326.684,Z 746.586,A -85,B 0,C 180,E1 -14966.858,E2 -14966.858} C_VEL
LIN {X 0,Y 326.635,Z 746.609,A -85,B 0,C 180,E1 -14970.61,E2 -14970.61} C_VEL
LIN {X 0,Y 326.608,Z 746.601,A -85,B 0,C 180,E1 -14974.019,E2 -14974.019} C_VEL
LIN {X 0,Y 326.628,Z 746.613,A -85,B 0,C 180,E1 -14977.239,E2 -14977.239} C_VEL
LIN {X 0,Y 326.578,Z 746.577,A -85,B 0,C 180,E1 -14981.131,E2 -14981.131} C_VEL
LIN {X 0,Y 326.528,Z 746.603,A -85,B 0,C 180,E1 -14984.743,E2 -14984.743} C_VEL
LIN {X 0,Y 326.577,Z 746.616,A -85,B 0,C 180,E1 -14988.154,E2 -14988.154} C_VEL
LIN {X 0,Y 326.599,Z 746.589,A -85,B 0,C 180,E1 -14991.388,E2 -14991.388} C_VEL
LIN {X 0,Y 326.621,Z 746.614,A -85,B 0,C 180,E1 -14994.851,E2 -14994.851} C_VEL
LIN {X 0,Y 326.609,Z 746.601,A -85,B 0,C 180,E1 -14997.456,E2 -14997.456} C_VEL
LIN {X 0,Y 326.618,Z 746.613,A -85,B 0,C 180,E1 -15000.337,E2 -15000.337} C_VEL
LIN {X 0,Y 326.644,Z 746.609,A -85,B 0,C 180,E1 -15004.644,E2 -15004.644} C_VEL
LIN {X 0,Y 326.686,Z 746.836,A -85,B 0,C 180,E1 -15007.05,E2 -15007.05} C_VEL
LIN {X 0,Y 327.76,Z 752.643,A -85,B 0,C 180,E1 -15009.28,E2 -15009.28} C_VEL
LIN {X 0,Y 328.101,Z 756.926,A -85,B 0,C 180,E1 -15010.771,E2 -15010.771} C_VEL
LIN {X 0,Y 328.822,Z 760.275,A -85,B 0,C 180,E1 -15010.957,E2 -15010.957} C_VEL
LIN {X 0,Y 332.886,Z 781.487,A -85,B 0,C 180,E1 -15011.675,E2 -15011.675} C_VEL
LIN {X 0,Y 332.082,Z 832.706,A -85,B 0,C 180,E1 -15012.805,E2 -15012.805} C_VEL
LIN {X 0,Y 331.827,Z 841.658,A -85,B 0,C 180,E1 -15013.148,E2 -15013.148} C_VEL
LIN {X 0,Y 331.264,Z 851.18,A -85,B 0,C 180,E1 -15013.674,E2 -15013.674} C_VEL
LIN {X 0,Y 330.687,Z 859.308,A -85,B 0,C 180,E1 -15014.278,E2 -15014.278} C_VEL
LIN {X 0,Y 329.858,Z 868.876,A -85,B 0,C 180,E1 -15015.186,E2 -15015.186} C_VEL
LIN {X 0,Y 328.955,Z 878.645,A -85,B 0,C 180,E1 -15016.408,E2 -15016.408} C_VEL
LIN {X 0,Y 328.103,Z 886.363,A -85,B 0,C 180,E1 -15017.631,E2 -15017.631} C_VEL
LIN {X 0,Y 327.347,Z 892.707,A -85,B 0,C 180,E1 -15018.859,E2 -15018.859} C_VEL
LIN {X 0,Y 326.705,Z 897.979,A -85,B 0,C 180,E1 -15020.09,E2 -15020.09} C_VEL
LIN {X 0,Y 326.219,Z 902.378,A -85,B 0,C 180,E1 -15021.326,E2 -15021.326} C_VEL
LIN {X 0,Y 325.742,Z 907.011,A -85,B 0,C 180,E1 -15022.963,E2 -15022.963} C_VEL
LIN {X 0,Y 325.437,Z 910.201,A -85,B 0,C 180,E1 -15024.423,E2 -15024.423} C_VEL
LIN {X 0,Y 325.094,Z 913.108,A -85,B 0,C 180,E1 -15026.281,E2 -15026.281} C_VEL
LIN {X 0,Y 324.954,Z 914.377,A -85,B 0,C 180,E1 -15027.521,E2 -15027.521} C_VEL
LIN {X 0,Y 324.88,Z 915.177,A -85,B 0,C 180,E1 -15028.76,E2 -15028.76} C_VEL
LIN {X 0,Y 324.879,Z 915.482,A -85,B 0,C 180,E1 -15030,E2 -15030} C_VEL
LIN {X 0,Y 324.878,Z 915.204,A -85,B 0,C 180,E1 -15031.24,E2 -15031.24} C_VEL
LIN {X 0,Y 324.944,Z 914.459,A -85,B 0,C 180,E1 -15032.479,E2 -15032.479} C_VEL
LIN {X 0,Y 325.092,Z 913.244,A -85,B 0,C 180,E1 -15033.719,E2 -15033.719} C_VEL
LIN {X 0,Y 325.423,Z 910.395,A -85,B 0,C 180,E1 -15035.577,E2 -15035.577} C_VEL
LIN {X 0,Y 325.728,Z 907.316,A -85,B 0,C 180,E1 -15037.016,E2 -15037.016} C_VEL
LIN {X 0,Y 326.147,Z 902.702,A -85,B 0,C 180,E1 -15038.676,E2 -15038.676} C_VEL
LIN {X 0,Y 326.806,Z 897.21,A -85,B 0,C 180,E1 -15040.219,E2 -15040.219} C_VEL
LIN {X 0,Y 327.675,Z 890.304,A -85,B 0,C 180,E1 -15041.757,E2 -15041.757} C_VEL
LIN {X 0,Y 328.595,Z 882.373,A -85,B 0,C 180,E1 -15043.135,E2 -15043.135} C_VEL
LIN {X 0,Y 329.384,Z 874.81,A -85,B 0,C 180,E1 -15044.204,E2 -15044.204} C_VEL
LIN {X 0,Y 330.035,Z 868.375,A -85,B 0,C 180,E1 -15044.963,E2 -15044.963} C_VEL
LIN {X 0,Y 330.679,Z 860.553,A -85,B 0,C 180,E1 -15045.723,E2 -15045.723} C_VEL
LIN {X 0,Y 331.33,Z 851.579,A -85,B 0,C 180,E1 -15046.402,E2 -15046.402} C_VEL
LIN {X 0,Y 331.788,Z 842.21,A -85,B 0,C 180,E1 -15046.933,E2 -15046.933} C_VEL
LIN {X 0,Y 332.065,Z 833.179,A -85,B 0,C 180,E1 -15047.287,E2 -15047.287} C_VEL
LIN {X 0,Y 332.791,Z 780.583,A -85,B 0,C 180,E1 -15048.457,E2 -15048.457} C_VEL
LIN {X 0,Y 328.561,Z 758.913,A -85,B 0,C 180,E1 -15049.197,E2 -15049.197} C_VEL
LIN {X 0,Y 328.071,Z 756.786,A -85,B 0,C 180,E1 -15049.312,E2 -15049.312} C_VEL
LIN {X 0,Y 327.533,Z 751.126,A -85,B 0,C 180,E1 -15051.394,E2 -15051.394} C_VEL
LIN {X 0,Y 326.721,Z 746.676,A -85,B 0,C 180,E1 -15053.198,E2 -15053.198} C_VEL
LIN {X 0,Y 326.616,Z 746.614,A -85,B 0,C 180,E1 -15056.864,E2 -15056.864} C_VEL
LIN {X 0,Y 326.613,Z 746.604,A -85,B 0,C 180,E1 -15060.603,E2 -15060.603} C_VEL
LIN {X 0,Y 326.608,Z 746.613,A -85,B 0,C 180,E1 -15064.019,E2 -15064.019} C_VEL
LIN {X 0,Y 326.628,Z 746.595,A -85,B 0,C 180,E1 -15067.238,E2 -15067.238} C_VEL
LIN {X 0,Y 326.598,Z 746.589,A -85,B 0,C 180,E1 -15068.664,E2 -15068.664} C_VEL
LIN {X 0,Y 325.932,Z 746.68,A -85,B 0,C 180,E1 -15069.692,E2 -15069.692} C_VEL
LIN {X 0,Y 323.066,Z 747.053,A -85,B 0,C 180,E1 -15071.365,E2 -15071.365} C_VEL
LIN {X 0,Y 320.628,Z 747.36,A -85,B 0,C 180,E1 -15072.721,E2 -15072.721} C_VEL
LIN {X 0,Y 319.575,Z 747.487,A -85,B 0,C 180,E1 -15073.771,E2 -15073.771} C_VEL
LIN {X 0,Y 319.485,Z 747.489,A -85,B 0,C 180,E1 -15074.127,E2 -15074.127} C_VEL
LIN {X 0,Y 319.554,Z 747.442,A -85,B 0,C 180,E1 -15077.016,E2 -15077.016} C_VEL
LIN {X 0,Y 319.548,Z 747.474,A -85,B 0,C 180,E1 -15080.371,E2 -15080.371} C_VEL
LIN {X 0,Y 319.56,Z 747.49,A -85,B 0,C 180,E1 -15083.572,E2 -15083.572} C_VEL
LIN {X 0,Y 319.578,Z 747.474,A -85,B 0,C 180,E1 -15086.686,E2 -15086.686} C_VEL
LIN {X 0,Y 319.586,Z 747.487,A -85,B 0,C 180,E1 -15089.616,E2 -15089.616} C_VEL
LIN {X 0,Y 319.607,Z 747.478,A -85,B 0,C 180,E1 -15092.498,E2 -15092.498} C_VEL
LIN {X 0,Y 319.604,Z 747.471,A -85,B 0,C 180,E1 -15095.304,E2 -15095.304} C_VEL
LIN {X 0,Y 319.6,Z 747.484,A -85,B 0,C 180,E1 -15099.4,E2 -15099.4} C_VEL
LIN {X 0,Y 319.626,Z 747.463,A -85,B 0,C 180,E1 -15102.071,E2 -15102.071} C_VEL
LIN {X 0,Y 319.734,Z 747.466,A -85,B 0,C 180,E1 -15106.008,E2 -15106.008} C_VEL
LIN {X 0,Y 319.759,Z 747.456,A -85,B 0,C 180,E1 -15109.873,E2 -15109.873} C_VEL
LIN {X 0,Y 319.934,Z 747.414,A -85,B 0,C 180,E1 -15112.426,E2 -15112.426} C_VEL
LIN {X 0,Y 319.749,Z 747.456,A -85,B 0,C 180,E1 -15114.956,E2 -15114.956} C_VEL
LIN {X 0,Y 320.01,Z 747.437,A -85,B 0,C 180,E1 -15117.482,E2 -15117.482} C_VEL
LIN {X 0,Y 320.151,Z 747.405,A -85,B 0,C 180,E1 -15120,E2 -15120} C_VEL
LIN {X 0,Y 319.991,Z 747.408,A -85,B 0,C 180,E1 -15122.517,E2 -15122.517} C_VEL
LIN {X 0,Y 319.945,Z 747.442,A -85,B 0,C 180,E1 -15126.305,E2 -15126.305} C_VEL
LIN {X 0,Y 319.839,Z 747.453,A -85,B 0,C 180,E1 -15128.848,E2 -15128.848} C_VEL
LIN {X 0,Y 319.683,Z 747.452,A -85,B 0,C 180,E1 -15132.7,E2 -15132.7} C_VEL
LIN {X 0,Y 319.701,Z 747.467,A -85,B 0,C 180,E1 -15135.295,E2 -15135.295} C_VEL
LIN {X 0,Y 319.678,Z 747.47,A -85,B 0,C 180,E1 -15139.255,E2 -15139.255} C_VEL
LIN {X 0,Y 319.574,Z 747.48,A -85,B 0,C 180,E1 -15143.319,E2 -15143.319} C_VEL
LIN {X 0,Y 319.635,Z 747.483,A -85,B 0,C 180,E1 -15146.088,E2 -15146.088} C_VEL
LIN {X 0,Y 319.58,Z 747.471,A -85,B 0,C 180,E1 -15148.934,E2 -15148.934} C_VEL
LIN {X 0,Y 319.532,Z 747.491,A -85,B 0,C 180,E1 -15151.862,E2 -15151.862} C_VEL
LIN {X 0,Y 319.582,Z 747.48,A -85,B 0,C 180,E1 -15155.543,E2 -15155.543} C_VEL
LIN {X 0,Y 319.582,Z 747.441,A -85,B 0,C 180,E1 -15158.007,E2 -15158.007} C_VEL
LIN {X 0,Y 319.569,Z 747.464,A -85,B 0,C 180,E1 -15161.606,E2 -15161.606} C_VEL
LIN {X 0,Y 319.503,Z 747.497,A -85,B 0,C 180,E1 -15165.26,E2 -15165.26} C_VEL
LIN {X 0,Y 319.528,Z 747.473,A -85,B 0,C 180,E1 -15168.712,E2 -15168.712} C_VEL
LIN {X 0,Y 319.579,Z 747.489,A -85,B 0,C 180,E1 -15172.344,E2 -15172.344} C_VEL
LIN {X 0,Y 319.561,Z 747.485,A -85,B 0,C 180,E1 -15175.123,E2 -15175.123} C_VEL
LIN {X 0,Y 319.57,Z 747.461,A -85,B 0,C 180,E1 -15179.058,E2 -15179.058} C_VEL
LIN {X 0,Y 319.655,Z 747.694,A -85,B 0,C 180,E1 -15181.629,E2 -15181.629} C_VEL
LIN {X 0,Y 321.647,Z 757.796,A -85,B 0,C 180,E1 -15185.127,E2 -15185.127} C_VEL
LIN {X 0,Y 322.202,Z 761.516,A -85,B 0,C 180,E1 -15186.365,E2 -15186.365} C_VEL
LIN {X 0,Y 321.675,Z 767.378,A -85,B 0,C 180,E1 -15188.197,E2 -15188.197} C_VEL
LIN {X 0,Y 320.961,Z 774.157,A -85,B 0,C 180,E1 -15190.239,E2 -15190.239} C_VEL
LIN {X 0,Y 321.533,Z 777.981,A -85,B 0,C 180,E1 -15190.436,E2 -15190.436} C_VEL
LIN {X 0,Y 325.007,Z 800.721,A -85,B 0,C 180,E1 -15191.171,E2 -15191.171} C_VEL
LIN {X 0,Y 325.825,Z 808.643,A -85,B 0,C 180,E1 -15191.4,E2 -15191.4} C_VEL
LIN {X 0,Y 325.129,Z 850.761,A -85,B 0,C 180,E1 -15192.351,E2 -15192.351} C_VEL
LIN {X 0,Y 324.705,Z 859.735,A -85,B 0,C 180,E1 -15192.686,E2 -15192.686} C_VEL
LIN {X 0,Y 324.092,Z 869.38,A -85,B 0,C 180,E1 -15193.221,E2 -15193.221} C_VEL
LIN {X 0,Y 323.398,Z 878.534,A -85,B 0,C 180,E1 -15193.914,E2 -15193.914} C_VEL
LIN {X 0,Y 322.359,Z 889.331,A -85,B 0,C 180,E1 -15194.995,E2 -15194.995} C_VEL
LIN {X 0,Y 321.261,Z 898.64,A -85,B 0,C 180,E1 -15196.237,E2 -15196.237} C_VEL
LIN {X 0,Y 320.464,Z 905.314,A -85,B 0,C 180,E1 -15197.332,E2 -15197.332} C_VEL
LIN {X 0,Y 319.742,Z 911.653,A -85,B 0,C 180,E1 -15198.59,E2 -15198.59} C_VEL
LIN {X 0,Y 319.165,Z 916.922,A -85,B 0,C 180,E1 -15199.854,E2 -15199.854} C_VEL
LIN {X 0,Y 318.673,Z 921.317,A -85,B 0,C 180,E1 -15201.119,E2 -15201.119} C_VEL
LIN {X 0,Y 318.201,Z 926.502,A -85,B 0,C 180,E1 -15203.023,E2 -15203.023} C_VEL
LIN {X 0,Y 317.9,Z 930.31,A -85,B 0,C 180,E1 -15204.927,E2 -15204.927} C_VEL
LIN {X 0,Y 317.849,Z 932.063,A -85,B 0,C 180,E1 -15206.197,E2 -15206.197} C_VEL
LIN {X 0,Y 317.766,Z 933.317,A -85,B 0,C 180,E1 -15207.465,E2 -15207.465} C_VEL
